Yaskawa INFORM job: DPRINT3D10.JBI

/JOB
//NAME DPRINT3D10
//POS
///NPOS 985,0,0,0,0,0
///TOOL 9
///POSTYPE PULSE
///PULSE
C00000=48313,52303,-120095,63672,-120169,-93276,0
C00001=48292,52332,-119999,63708,-120197,-93246,0
C00002=48271,52372,-119870,63749,-120237,-93206,0
C00003=48256,52403,-119767,63780,-120271,-93175,0
C00004=48247,52435,-119662,63805,-120306,-93144,0
C00005=48242,52474,-119535,63828,-120351,-93108,0
C00006=48240,52507,-119427,63845,-120390,-93077,0
C00007=48244,52540,-119319,63857,-120432,-93047,0
C00008=48254,52576,-119202,63863,-120480,-93015,0
C00009=48265,52610,-119093,63867,-120523,-92986,0
C00010=48282,52644,-118984,63864,-120571,-92958,0
C00011=48286,52651,-118962,63862,-120581,-92952,0
C00012=48302,52701,-118799,63868,-120646,-92909,0
C00013=30148,51851,-121170,60929,-120456,-93852,0
C00014=30162,51845,-121190,60911,-120453,-93859,0
C00015=30223,51818,-121280,60832,-120438,-93894,0
C00016=30294,51784,-121396,60738,-120418,-93935,0
C00017=30355,51745,-121525,60652,-120388,-93980,0
C00018=30411,51705,-121661,60572,-120352,-94026,0
C00019=30455,51662,-121806,60503,-120310,-94072,0
C00020=30494,51618,-121956,60440,-120263,-94119,0
C00021=30520,51571,-122113,60390,-120209,-94166,0
C00022=30539,51524,-122271,60346,-120151,-94213,0
C00023=30546,51477,-122432,60317,-120088,-94259,0
C00024=30545,51429,-122594,60295,-120021,-94303,0
C00025=30531,51382,-122754,60288,-119952,-94345,0
C00026=30511,51335,-122911,60290,-119880,-94386,0
C00027=30478,51291,-123064,60306,-119806,-94423,0
C00028=30438,51247,-123212,60330,-119733,-94459,0
C00029=30386,51206,-123350,60368,-119658,-94491,0
C00030=30328,51167,-123484,60415,-119583,-94519,0
C00031=30311,51158,-123514,60429,-119566,-94525,0
C00032=30263,51130,-123609,60469,-119511,-94545,0
C00033=30203,51101,-123709,60523,-119450,-94565,0
C00034=30111,51065,-123831,60608,-119369,-94586,0
C00035=30037,51041,-123911,60678,-119311,-94599,0
C00036=29931,51014,-124003,60783,-119238,-94610,0
C00037=29846,50997,-124062,60869,-119186,-94615,0
C00038=29731,50980,-124118,60989,-119124,-94615,0
C00039=29637,50970,-124150,61088,-119080,-94611,0
C00040=29518,50964,-124170,61217,-119032,-94601,0
C00041=29419,50962,-124173,61325,-118997,-94589,0
C00042=29301,50967,-124156,61458,-118964,-94568,0
C00043=29202,50974,-124127,61570,-118942,-94547,0
C00044=29088,50989,-124074,61703,-118925,-94516,0
C00045=29047,50995,-124051,61750,-118920,-94505,0
C00046=28992,51005,-124016,61816,-118916,-94487,0
C00047=28937,51018,-123970,61882,-118916,-94467,0
C00048=28868,51035,-123909,61966,-118916,-94441,0
C00049=28800,51055,-123840,62049,-118920,-94412,0
C00050=28711,51089,-123723,62163,-118936,-94367,0
C00051=28673,51104,-123669,62211,-118944,-94346,0
C00052=28632,51124,-123601,62266,-118957,-94322,0
C00053=28562,51163,-123464,62360,-118987,-94274,0
C00054=28530,51183,-123394,62404,-119003,-94249,0
C00055=28500,51205,-123319,62448,-119023,-94224,0
C00056=28479,51224,-123254,62479,-119041,-94203,0
C00057=28453,51251,-123161,62520,-119069,-94173,0
C00058=28414,51299,-122996,62585,-119119,-94121,0
C00059=28390,51349,-122825,62634,-119177,-94069,0
C00060=28372,51400,-122652,62677,-119238,-94017,0
C00061=28369,51452,-122476,62703,-119305,-93967,0
C00062=28374,51504,-122300,62722,-119375,-93918,0
C00063=28378,51516,-122258,62723,-119393,-93907,0
C00064=28393,51556,-122125,62724,-119449,-93871,0
C00065=28418,51607,-121954,62719,-119525,-93826,0
C00066=28461,51656,-121791,62695,-119603,-93786,0
C00067=28512,51703,-121635,62661,-119681,-93749,0
C00068=28543,51726,-121555,62637,-119724,-93731,0
C00069=28573,51746,-121489,62613,-119760,-93717,0
C00070=28645,51790,-121346,62555,-119842,-93686,0
C00071=28701,51817,-121255,62506,-119897,-93669,0
C00072=28759,51842,-121173,62453,-119950,-93654,0
C00073=28805,51861,-121111,62411,-119991,-93643,0
C00074=28853,51877,-121058,62366,-120029,-93635,0
C00075=28890,51889,-121021,62331,-120057,-93630,0
C00076=28990,51916,-120931,62234,-120128,-93618,0
C00077=29081,51935,-120870,62143,-120186,-93614,0
C00078=29190,51953,-120814,62031,-120248,-93614,0
C00079=29284,51962,-120783,61932,-120294,-93620,0
C00080=29399,51970,-120761,61809,-120344,-93630,0
C00081=29492,51970,-120760,61707,-120379,-93643,0
C00082=29608,51966,-120775,61579,-120415,-93664,0
C00083=29697,51959,-120803,61477,-120437,-93685,0
C00084=29810,51944,-120856,61345,-120458,-93715,0
C00085=29891,51928,-120908,61248,-120467,-93742,0
C00086=29997,51902,-120995,61120,-120471,-93782,0
C00087=30066,51881,-121068,61034,-120467,-93812,0
C00088=30146,51842,-121200,60928,-120443,-93860,0
C00089=25451,55201,-110574,67596,-122310,-90184,0
C00090=36364,52150,-120303,76476,-115314,-91905,0
C00091=38692,59001,-99858,76810,-121576,-86102,0
C00092=38615,59038,-99753,76902,-121554,-86062,0
C00093=38581,59057,-99701,76944,-121546,-86041,0
C00094=38542,59080,-99635,76993,-121538,-86017,0
C00095=38475,59130,-99497,77080,-121530,-85968,0
C00096=38443,59156,-99424,77123,-121528,-85943,0
C00097=38413,59183,-99346,77165,-121528,-85916,0
C00098=38391,59209,-99275,77197,-121531,-85893,0
C00099=38362,59245,-99174,77242,-121537,-85860,0
C00100=38317,59310,-98994,77314,-121551,-85802,0
C00101=38282,59379,-98800,77378,-121575,-85741,0
C00102=38253,59451,-98602,77437,-121602,-85680,0
C00103=38236,59525,-98397,77486,-121639,-85618,0
C00104=38224,59600,-98189,77530,-121679,-85557,0
C00105=38224,59618,-98139,77538,-121691,-85542,0
C00106=38225,59676,-97978,77562,-121728,-85496,0
C00107=38231,59753,-97768,77589,-121778,-85437,0
C00108=38251,59828,-97562,77602,-121838,-85380,0
C00109=38278,59901,-97362,77607,-121900,-85326,0
C00110=38297,59938,-97259,77605,-121935,-85300,0
C00111=38315,59970,-97171,77601,-121966,-85277,0
C00112=38360,60041,-96979,77587,-122037,-85228,0
C00113=38398,60086,-96854,77571,-122089,-85198,0
C00114=38438,60129,-96738,77550,-122139,-85170,0
C00115=38469,60162,-96650,77534,-122179,-85149,0
C00116=38503,60190,-96572,77514,-122218,-85131,0
C00117=38529,60211,-96516,77497,-122247,-85119,0
C00118=38602,60262,-96378,77448,-122323,-85090,0
C00119=38669,60299,-96278,77399,-122389,-85071,0
C00120=38752,60337,-96176,77335,-122463,-85053,0
C00121=38825,60362,-96109,77275,-122524,-85044,0
C00122=38914,60385,-96048,77198,-122594,-85039,0
C00123=38988,60396,-96017,77131,-122647,-85042,0
C00124=39082,60404,-95999,77043,-122710,-85050,0
C00125=39155,60403,-96003,76971,-122755,-85061,0
C00126=39249,60394,-96030,76875,-122808,-85083,0
C00127=39319,60380,-96067,76801,-122842,-85104,0
C00128=39410,60355,-96138,76701,-122883,-85137,0
C00129=39473,60331,-96204,76628,-122907,-85165,0
C00130=39557,60290,-96318,76527,-122932,-85210,0
C00131=39612,60258,-96406,76459,-122946,-85243,0
C00132=39678,60217,-96522,76375,-122960,-85286,0
C00133=39737,60168,-96657,76295,-122964,-85333,0
C00134=39792,60116,-96800,76218,-122964,-85382,0
C00135=39839,60058,-96960,76145,-122955,-85434,0
C00136=39881,59998,-97125,76076,-122941,-85488,0
C00137=39915,59933,-97303,76014,-122919,-85544,0
C00138=39943,59868,-97485,75956,-122893,-85600,0
C00139=39961,59799,-97674,75907,-122859,-85657,0
C00140=39974,59730,-97865,75863,-122821,-85713,0
C00141=39976,59660,-98058,75829,-122776,-85769,0
C00142=39973,59590,-98250,75801,-122728,-85823,0
C00143=39959,59521,-98440,75783,-122672,-85875,0
C00144=39940,59453,-98627,75772,-122616,-85926,0
C00145=39910,59389,-98806,75772,-122555,-85973,0
C00146=39875,59325,-98980,75778,-122492,-86018,0
C00147=39865,59311,-99021,75782,-122476,-86028,0
C00148=39835,59265,-99148,75791,-122426,-86060,0
C00149=39795,59216,-99283,75809,-122370,-86093,0
C00150=39733,59154,-99454,75843,-122292,-86133,0
C00151=39682,59111,-99571,75875,-122233,-86159,0
C00152=39606,59061,-99711,75928,-122154,-86188,0
C00153=39543,59026,-99805,75975,-122094,-86206,0
C00154=39457,58990,-99905,76045,-122018,-86223,0
C00155=39386,58966,-99971,76105,-121961,-86232,0
C00156=39293,58944,-100030,76188,-121892,-86236,0
C00157=39216,58931,-100063,76259,-121838,-86235,0
C00158=39120,58925,-100079,76352,-121777,-86225,0
C00159=39039,58925,-100077,76432,-121730,-86214,0
C00160=38945,58934,-100049,76530,-121681,-86192,0
C00161=38911,58939,-100035,76566,-121665,-86184,0
C00162=38864,58948,-100010,76617,-121642,-86170,0
C00163=38816,58961,-99973,76669,-121622,-86152,0
C00164=38771,58974,-99936,76720,-121604,-86136,0
C00165=38691,59038,-99755,76827,-121599,-86073,0
C00166=38691,58985,-99777,76837,-121614,-86054,0
C00167=29066,51891,-120835,62177,-120230,-93576,0
C00168=29144,51906,-120784,62099,-120279,-93573,0
C00169=29192,51914,-120759,62050,-120306,-93573,0
C00170=29275,51924,-120728,61964,-120349,-93577,0
C00171=29382,51934,-120697,61850,-120400,-93584,0
C00172=29408,51935,-120694,61823,-120411,-93587,0
C00173=29492,51937,-120689,61731,-120443,-93597,0
C00174=29601,51937,-120692,61611,-120483,-93614,0
C00175=29709,51929,-120719,61488,-120512,-93637,0
C00176=29816,51918,-120756,61365,-120536,-93663,0
C00177=29841,51915,-120769,61337,-120541,-93670,0
C00178=29919,51901,-120815,61244,-120551,-93694,0
C00179=29968,51891,-120850,61186,-120554,-93711,0
C00180=30019,51879,-120890,61124,-120558,-93729,0
C00181=30067,51865,-120937,61065,-120557,-93750,0
C00182=30111,51851,-120985,61010,-120553,-93769,0
C00183=30201,51818,-121097,60894,-120542,-93813,0
C00184=30258,51792,-121184,60819,-120527,-93846,0
C00185=30312,51764,-121277,60747,-120510,-93880,0
C00186=30351,51743,-121349,60694,-120495,-93905,0
C00187=30385,51721,-121422,60647,-120477,-93930,0
C00188=30409,51703,-121483,60612,-120461,-93950,0
C00189=30472,51651,-121655,60518,-120414,-94007,0
C00190=30501,51621,-121759,60472,-120383,-94040,0
C00191=30527,51587,-121870,60428,-120346,-94075,0
C00192=30547,51560,-121964,60393,-120317,-94103,0
C00193=30561,51532,-122059,60364,-120283,-94131,0
C00194=30576,51489,-122201,60329,-120230,-94173,0
C00195=30584,51460,-122300,60306,-120192,-94202,0
C00196=30586,51430,-122400,60289,-120153,-94229,0
C00197=30583,51390,-122537,60274,-120097,-94267,0
C00198=30579,51360,-122638,60265,-120053,-94294,0
C00199=30569,51330,-122740,60262,-120009,-94321,0
C00200=30549,51293,-122864,60267,-119951,-94352,0
C00201=30532,51263,-122965,60273,-119904,-94377,0
C00202=30508,51234,-123063,60285,-119856,-94401,0
C00203=30475,51202,-123172,60306,-119801,-94427,0
C00204=30445,51174,-123266,60327,-119751,-94449,0
C00205=30408,51147,-123358,60356,-119701,-94469,0
C00206=30365,51121,-123448,60391,-119650,-94488,0
C00207=30321,51096,-123533,60428,-119601,-94506,0
C00208=30272,51072,-123615,60471,-119550,-94521,0
C00209=30185,51035,-123739,60550,-119471,-94544,0
C00210=30103,51007,-123835,60629,-119403,-94560,0
C00211=30015,50981,-123923,60713,-119339,-94572,0
C00212=29922,50960,-123992,60807,-119279,-94579,0
C00213=29825,50943,-124051,60906,-119221,-94582,0
C00214=29724,50931,-124089,61012,-119172,-94579,0
C00215=29622,50922,-124118,61121,-119126,-94574,0
C00216=29518,50919,-124126,61235,-119088,-94561,0
C00217=29414,50920,-124123,61350,-119054,-94547,0
C00218=29311,50926,-124098,61466,-119030,-94526,0
C00219=29209,50936,-124063,61583,-119009,-94503,0
C00220=29112,50951,-124009,61697,-118997,-94474,0
C00221=29017,50969,-123943,61810,-118992,-94443,0
C00222=28929,50993,-123859,61918,-118995,-94408,0
C00223=28844,51020,-123766,62023,-119002,-94370,0
C00224=28758,51055,-123643,62134,-119021,-94324,0
C00225=28707,51078,-123564,62201,-119035,-94294,0
C00226=28662,51102,-123481,62261,-119053,-94265,0
C00227=28618,51127,-123394,62320,-119071,-94234,0
C00228=28580,51153,-123304,62374,-119093,-94204,0
C00229=28548,51181,-123210,62422,-119119,-94173,0
C00230=28514,51211,-123106,62473,-119148,-94138,0
C00231=28489,51240,-123007,62514,-119178,-94107,0
C00232=28469,51269,-122907,62548,-119210,-94076,0
C00233=28448,51305,-122785,62587,-119250,-94039,0
C00234=28437,51335,-122684,62614,-119285,-94008,0
C00235=28431,51365,-122582,62634,-119323,-93979,0
C00236=28425,51404,-122448,62658,-119372,-93941,0
C00237=28426,51434,-122347,62671,-119412,-93912,0
C00238=28433,51464,-122247,62677,-119454,-93884,0
C00239=28445,51506,-122106,62683,-119512,-93847,0
C00240=28458,51534,-122012,62681,-119554,-93822,0
C00241=28477,51563,-121915,62673,-119597,-93797,0
C00242=28507,51605,-121775,62659,-119663,-93761,0
C00243=28531,51631,-121688,62645,-119705,-93740,0
C00244=28561,51657,-121601,62624,-119749,-93720,0
C00245=28599,51689,-121496,62597,-119803,-93696,0
C00246=28643,51721,-121390,62563,-119860,-93672,0
C00247=28717,51764,-121249,62502,-119942,-93643,0
C00248=28750,51781,-121192,62474,-119975,-93632,0
C00249=28790,51800,-121130,62439,-120014,-93620,0
C00250=28836,51818,-121070,62396,-120055,-93609,0
C00251=28900,51842,-120990,62338,-120109,-93596,0
C00252=28965,51864,-120920,62276,-120160,-93585,0
C00253=28974,51867,-120912,62267,-120166,-93585,0
C00254=29068,51902,-120798,62180,-120245,-93566,0
C00255=39943,50914,-124372,72212,-115599,-93497,0
C00256=35334,54043,-114097,78273,-116418,-89868,0
C00257=36297,54454,-112860,77429,-117185,-89597,0
C00258=40949,51295,-123088,71276,-116378,-93209,0
C00259=40026,50945,-124269,72134,-115663,-93473,0
C00260=35605,54738,-111986,78248,-117048,-89258,0
C00261=36478,55133,-110816,77500,-117769,-89005,0
C00262=42177,51262,-123232,69935,-116794,-93388,0
C00263=33602,54748,-111917,58580,-125515,-91919,0
C00264=34233,54163,-113709,79451,-115969,-89637,0
C00265=35135,54535,-112592,78656,-116671,-89391,0
C00266=34900,54747,-111946,78974,-116702,-89171,0
C00267=35368,54950,-111341,78569,-117079,-89039,0
C00268=35551,54786,-111840,78321,-117055,-89209,0
C00269=36110,54506,-112698,77641,-117132,-89528,0
C00270=34834,55007,-111160,57349,-126335,-91958,0
C00271=36863,53301,-116438,54206,-124911,-93686,0
C00272=39303,53272,-116584,73829,-117628,-91057,0
C00273=44071,55812,-108960,69905,-122100,-89467,0
C00274=34853,54989,-111215,79109,-116844,-88946,0
C00275=33011,56887,-105605,81638,-117037,-87071,0
C00276=36074,54033,-114146,77503,-116763,-89961,0
C00277=40139,51272,-123147,72141,-116051,-93140,0
C00278=48385,52777,-118383,63852,-120867,-92777,0
C00279=48412,52795,-118324,63830,-120899,-92765,0
C00280=48487,52840,-118184,63770,-120980,-92737,0
C00281=48544,52867,-118098,63720,-121034,-92721,0
C00282=48600,52891,-118023,63670,-121084,-92709,0
C00283=48648,52910,-117962,63626,-121126,-92699,0
C00284=48698,52927,-117910,63579,-121165,-92691,0
C00285=48776,52949,-117842,63505,-121220,-92684,0
C00286=48831,52963,-117798,63452,-121258,-92680,0
C00287=48887,52975,-117762,63396,-121293,-92678,0
C00288=48966,52987,-117724,63315,-121339,-92680,0
C00289=49026,52996,-117698,63254,-121373,-92681,0
C00290=49087,53002,-117682,63189,-121403,-92686,0
C00291=49164,53006,-117671,63107,-121437,-92695,0
C00292=49227,53008,-117665,63039,-121465,-92703,0
C00293=49291,53007,-117669,62969,-121488,-92713,0
C00294=49363,53003,-117684,62888,-121511,-92728,0
C00295=49427,52999,-117699,62816,-121530,-92742,0
C00296=49490,52991,-117725,62743,-121545,-92759,0
C00297=49555,52981,-117761,62667,-121557,-92779,0
C00298=49617,52970,-117799,62593,-121567,-92799,0
C00299=49678,52955,-117846,62519,-121574,-92822,0
C00300=49777,52928,-117936,62398,-121578,-92861,0
C00301=49856,52900,-118025,62298,-121575,-92898,0
C00302=49946,52864,-118146,62182,-121563,-92945,0
C00303=50004,52833,-118246,62103,-121548,-92982,0
C00304=50069,52795,-118370,62013,-121525,-93026,0
C00305=50124,52753,-118507,61933,-121493,-93072,0
C00306=50173,52709,-118650,61858,-121458,-93119,0
C00307=50211,52662,-118802,61794,-121414,-93167,0
C00308=50244,52614,-118958,61735,-121366,-93215,0
C00309=50263,52564,-119119,61690,-121311,-93263,0
C00310=50277,52514,-119283,61651,-121252,-93310,0
C00311=50277,52463,-119448,61626,-121189,-93356,0
C00312=50272,52413,-119612,61609,-121122,-93400,0
C00313=50253,52363,-119773,61606,-121053,-93442,0
C00314=50228,52314,-119932,61611,-120982,-93482,0
C00315=50186,52261,-120104,61632,-120899,-93523,0
C00316=50157,52229,-120210,61649,-120847,-93548,0
C00317=50124,52200,-120306,61671,-120798,-93570,0
C00318=50088,52170,-120403,61696,-120748,-93592,0
C00319=50049,52143,-120491,61726,-120698,-93611,0
C00320=50006,52117,-120574,61763,-120650,-93627,0
C00321=49957,52090,-120662,61804,-120598,-93645,0
C00322=49908,52067,-120736,61847,-120551,-93658,0
C00323=49856,52047,-120800,61895,-120507,-93669,0
C00324=49793,52024,-120876,61954,-120454,-93681,0
C00325=49737,52007,-120930,62007,-120413,-93688,0
C00326=49680,51993,-120976,62064,-120374,-93692,0
C00327=49604,51975,-121033,62139,-120326,-93697,0
C00328=49545,51964,-121067,62199,-120290,-93698,0
C00329=49483,51956,-121092,62263,-120258,-93697,0
C00330=49397,51946,-121124,62353,-120214,-93693,0
C00331=49337,51941,-121138,62417,-120188,-93689,0
C00332=49275,51939,-121144,62484,-120163,-93681,0
C00333=49182,51937,-121147,62586,-120128,-93669,0
C00334=49123,51938,-121142,62651,-120109,-93659,0
C00335=49063,51942,-121127,62719,-120093,-93646,0
C00336=48988,51948,-121106,62804,-120073,-93630,0
C00337=48912,51956,-121075,62892,-120057,-93610,0
C00338=48805,51975,-121011,63018,-120042,-93577,0
C00339=48760,51984,-120980,63071,-120037,-93562,0
C00340=48707,51997,-120936,63136,-120035,-93542,0
C00341=48615,52024,-120843,63249,-120036,-93503,0
C00342=48572,52038,-120793,63303,-120038,-93483,0
C00343=48528,52055,-120737,63360,-120043,-93461,0
C00344=48453,52089,-120622,63457,-120059,-93418,0
C00345=48394,52123,-120512,63537,-120079,-93379,0
C00346=48365,52142,-120445,63579,-120093,-93356,0
C00347=48320,52178,-120328,63644,-120120,-93316,0
C00348=48268,52225,-120171,63723,-120159,-93265,0
C00349=48259,52237,-120133,63739,-120169,-93252,0
C00350=48230,52276,-120004,63788,-120206,-93212,0
C00351=48197,52328,-119833,63848,-120258,-93159,0
C00352=48180,52381,-119657,63892,-120317,-93107,0
C00353=48169,52436,-119478,63930,-120379,-93054,0
C00354=48169,52449,-119435,63935,-120395,-93043,0
C00355=48172,52491,-119298,63952,-120446,-93005,0
C00356=48177,52518,-119212,63958,-120480,-92981,0
C00357=48185,52546,-119120,63963,-120517,-92956,0
C00358=48198,52574,-119031,63961,-120556,-92933,0
C00359=48213,52600,-118947,63957,-120591,-92911,0
C00360=48250,52655,-118771,63942,-120672,-92867,0
C00361=48284,52691,-118655,63922,-120727,-92839,0
C00362=48322,52727,-118542,63897,-120783,-92813,0
C00363=48328,52732,-118524,63893,-120792,-92809,0
C00364=48363,52780,-118371,63877,-120862,-92771,0
C00365=39595,59020,-99695,75955,-122172,-86157,0
C00366=39524,58985,-99793,76010,-122107,-86175,0
C00367=39448,58957,-99869,76074,-122043,-86186,0
C00368=39369,58933,-99934,76141,-121981,-86194,0
C00369=39287,58918,-99974,76216,-121923,-86194,0
C00370=39205,58907,-100002,76293,-121867,-86190,0
C00371=39121,58906,-100005,76376,-121816,-86179,0
C00372=39038,58909,-99994,76460,-121769,-86165,0
C00373=38956,58921,-99960,76547,-121729,-86143,0
C00374=38875,58937,-99913,76634,-121692,-86119,0
C00375=38798,58962,-99841,76721,-121663,-86087,0
C00376=38723,58991,-99759,76808,-121638,-86053,0
C00377=38644,59033,-99641,76905,-121617,-86008,0
C00378=38596,59061,-99563,76964,-121607,-85979,0
C00379=38554,59090,-99480,77019,-121601,-85950,0
C00380=38512,59122,-99392,77074,-121597,-85918,0
C00381=38474,59155,-99299,77126,-121596,-85886,0
C00382=38440,59191,-99198,77175,-121598,-85853,0
C00383=38404,59231,-99087,77227,-121602,-85816,0
C00384=38375,59270,-98979,77273,-121609,-85780,0
C00385=38351,59310,-98867,77313,-121621,-85745,0
C00386=38324,59359,-98731,77361,-121636,-85702,0
C00387=38306,59401,-98616,77397,-121651,-85667,0
C00388=38292,59444,-98497,77429,-121670,-85631,0
C00389=38276,59500,-98342,77468,-121696,-85584,0
C00390=38269,59542,-98224,77494,-121717,-85549,0
C00391=38266,59586,-98103,77516,-121744,-85513,0
C00392=38263,59647,-97934,77545,-121781,-85465,0
C00393=38265,59690,-97818,77561,-121808,-85432,0
C00394=38273,59733,-97699,77573,-121839,-85398,0
C00395=38285,59797,-97524,77588,-121886,-85350,0
C00396=38297,59837,-97413,77594,-121919,-85320,0
C00397=38313,59878,-97302,77596,-121954,-85290,0
C00398=38334,59928,-97165,77597,-121998,-85253,0
C00399=38361,59978,-97027,77593,-122046,-85217,0
C00400=38408,60048,-96836,77577,-122118,-85169,0
C00401=38430,60077,-96759,77568,-122149,-85150,0
C00402=38457,60108,-96673,77556,-122185,-85129,0
C00403=38489,60140,-96587,77539,-122225,-85109,0
C00404=38533,60182,-96473,77514,-122278,-85083,0
C00405=38579,60221,-96368,77485,-122331,-85059,0
C00406=38653,60270,-96235,77436,-122407,-85032,0
C00407=38711,60301,-96151,77393,-122462,-85015,0
C00408=38747,60318,-96106,77365,-122495,-85008,0
C00409=38811,60341,-96042,77313,-122549,-84999,0
C00410=38894,60368,-95971,77244,-122618,-84990,0
C00411=38914,60372,-95960,77226,-122633,-84990,0
C00412=38981,60384,-95928,77167,-122683,-84990,0
C00413=39068,60397,-95897,77087,-122745,-84994,0
C00414=39157,60398,-95894,77001,-122801,-85006,0
C00415=39245,60395,-95905,76914,-122854,-85022,0
C00416=39266,60392,-95913,76892,-122864,-85028,0
C00417=39332,60381,-95943,76823,-122899,-85046,0
C00418=39373,60372,-95969,76778,-122918,-85060,0
C00419=39417,60361,-96001,76730,-122939,-85075,0
C00420=39459,60346,-96042,76682,-122955,-85093,0
C00421=39498,60330,-96086,76637,-122969,-85111,0
C00422=39579,60293,-96190,76541,-122995,-85152,0
C00423=39631,60261,-96277,76475,-123008,-85185,0
C00424=39681,60227,-96371,76411,-123017,-85219,0
C00425=39718,60201,-96443,76363,-123023,-85245,0
C00426=39750,60173,-96520,76319,-123025,-85272,0
C00427=39775,60150,-96584,76284,-123025,-85294,0
C00428=39839,60082,-96770,76191,-123021,-85356,0
C00429=39870,60041,-96885,76141,-123013,-85393,0
C00430=39899,59996,-97009,76092,-123001,-85433,0
C00431=39922,59957,-97114,76051,-122990,-85467,0
C00432=39942,59919,-97221,76015,-122976,-85500,0
C00433=39964,59859,-97386,75965,-122950,-85550,0
C00434=39979,59817,-97501,75932,-122932,-85586,0
C00435=39989,59774,-97618,75902,-122910,-85621,0
C00436=39998,59715,-97780,75867,-122876,-85668,0
C00437=40003,59671,-97902,75842,-122849,-85704,0
C00438=40003,59626,-98026,75822,-122821,-85739,0
C00439=39998,59571,-98178,75802,-122780,-85781,0
C00440=39992,59526,-98303,75787,-122747,-85816,0
C00441=39981,59481,-98426,75778,-122710,-85850,0
C00442=39964,59431,-98564,75772,-122667,-85887,0
C00443=39948,59387,-98685,75768,-122628,-85920,0
C00444=39927,59344,-98804,75770,-122586,-85950,0
C00445=39900,59301,-98922,75777,-122541,-85980,0
C00446=39873,59260,-99036,75786,-122498,-86009,0
C00447=39841,59220,-99146,75800,-122452,-86036,0
C00448=39783,59157,-99318,75830,-122375,-86077,0
C00449=39725,59107,-99456,75864,-122307,-86108,0
C00450=39665,59062,-99582,75903,-122241,-86135,0
C00451=39599,58976,-99818,75931,-122145,-86193,0
C00452=23775,60523,-95311,71968,-125942,-85610,0
C00453=23816,60447,-95518,71888,-125912,-85675,0
C00454=23839,60389,-95677,71836,-125882,-85723,0
C00455=23861,60320,-95866,71779,-125844,-85780,0
C00456=23873,60249,-96060,71731,-125798,-85836,0
C00457=23879,60177,-96256,71689,-125749,-85892,0
C00458=23875,60105,-96451,71657,-125693,-85946,0
C00459=23866,60034,-96646,71631,-125634,-85998,0
C00460=23846,59965,-96835,71616,-125571,-86048,0
C00461=23820,59897,-97020,71608,-125504,-86095,0
C00462=23785,59833,-97196,71611,-125435,-86138,0
C00463=23745,59771,-97365,71621,-125365,-86179,0
C00464=23696,59715,-97521,71642,-125292,-86214,0
C00465=23643,59661,-97668,71669,-125221,-86246,0
C00466=23574,59607,-97815,71712,-125140,-86276,0
C00467=23529,59575,-97902,71742,-125089,-86293,0
C00468=23450,59528,-98030,71799,-125007,-86315,0
C00469=23388,59499,-98110,71847,-124949,-86327,0
C00470=23299,59467,-98198,71921,-124873,-86337,0
C00471=23230,59448,-98249,71982,-124818,-86340,0
C00472=23135,59432,-98293,72069,-124750,-86337,0
C00473=23061,59424,-98312,72140,-124701,-86330,0
C00474=22966,59424,-98311,72236,-124645,-86314,0
C00475=22889,59430,-98295,72316,-124604,-86297,0
C00476=22797,59446,-98249,72417,-124562,-86269,0
C00477=22721,59465,-98197,72502,-124532,-86242,0
C00478=22635,59496,-98109,72604,-124503,-86203,0
C00479=22563,59528,-98020,72691,-124485,-86167,0
C00480=22487,59573,-97895,72790,-124472,-86119,0
C00481=22458,59592,-97843,72828,-124470,-86099,0
C00482=22423,59618,-97772,72875,-124467,-86074,0
C00483=22389,59648,-97688,72924,-124468,-86045,0
C00484=22346,59688,-97578,72986,-124472,-86007,0
C00485=22306,59731,-97459,73047,-124480,-85967,0
C00486=22257,59798,-97273,73129,-124498,-85907,0
C00487=22236,59830,-97186,73165,-124510,-85878,0
C00488=22216,59866,-97087,73203,-124522,-85848,0
C00489=22186,59934,-96900,73265,-124554,-85790,0
C00490=22167,59996,-96731,73314,-124586,-85740,0
C00491=22160,60031,-96635,73338,-124606,-85711,0
C00492=22152,60091,-96471,73375,-124645,-85664,0
C00493=22147,60169,-96257,73417,-124697,-85603,0
C00494=22149,60187,-96208,73425,-124711,-85589,0
C00495=22155,60247,-96044,73448,-124757,-85544,0
C00496=22167,60325,-95832,73473,-124820,-85486,0
C00497=22192,60401,-95625,73486,-124888,-85432,0
C00498=22221,60475,-95423,73493,-124959,-85380,0
C00499=22230,60492,-95377,73492,-124976,-85368,0
C00500=22261,60546,-95231,73488,-125033,-85332,0
C00501=22283,60579,-95141,73482,-125069,-85311,0
C00502=22308,60613,-95049,73474,-125109,-85289,0
C00503=22336,60645,-94962,73461,-125149,-85269,0
C00504=22365,60674,-94884,73447,-125187,-85252,0
C00505=22429,60733,-94725,73413,-125267,-85217,0
C00506=22478,60769,-94627,73383,-125323,-85198,0
C00507=22529,60803,-94537,73348,-125379,-85181,0
C00508=22569,60827,-94472,73321,-125420,-85170,0
C00509=22608,60847,-94418,73292,-125458,-85161,0
C00510=22625,60855,-94398,73279,-125474,-85158,0
C00511=22680,60877,-94337,73236,-125523,-85151,0
C00512=22725,60895,-94291,73200,-125564,-85145,0
C00513=22769,60908,-94256,73163,-125600,-85143,0
C00514=22801,60915,-94236,73135,-125626,-85143,0
C00515=22890,60933,-94190,73055,-125693,-85144,0
C00516=22967,60940,-94172,72982,-125746,-85152,0
C00517=23059,60941,-94170,72892,-125804,-85167,0
C00518=23134,60934,-94190,72814,-125845,-85186,0
C00519=23224,60918,-94233,72716,-125890,-85213,0
C00520=23295,60899,-94286,72637,-125920,-85240,0
C00521=23381,60867,-94374,72534,-125951,-85279,0
C00522=23444,60837,-94457,72457,-125967,-85314,0
C00523=23522,60790,-94585,72355,-125982,-85363,0
C00524=23576,60750,-94693,72281,-125987,-85402,0
C00525=23644,60689,-94858,72183,-125983,-85460,0
C00526=23680,60651,-94963,72128,-125977,-85496,0
C00527=23732,60587,-95137,72043,-125962,-85553,0
C00528=23825,60523,-95313,71917,-125973,-85619,0
C00529=25489,55155,-110561,67572,-122361,-90161,0
C00530=36365,52089,-120325,76484,-115334,-91883,0
C00531=36365,52027,-120346,76491,-115352,-91861,0
C00532=23826,60495,-95267,71941,-126008,-85582,0
C00533=23863,60420,-95471,71866,-125976,-85646,0
C00534=23883,60366,-95619,71819,-125947,-85690,0
C00535=23897,60314,-95762,71778,-125918,-85733,0
C00536=23908,60271,-95878,71746,-125892,-85767,0
C00537=23914,60229,-95993,71718,-125865,-85801,0
C00538=23917,60163,-96173,71681,-125818,-85851,0
C00539=23918,60119,-96294,71658,-125785,-85885,0
C00540=23915,60075,-96412,71640,-125751,-85918,0
C00541=23904,60014,-96580,71620,-125698,-85963,0
C00542=23895,59969,-96701,71607,-125660,-85995,0
C00543=23881,59926,-96819,71599,-125619,-86026,0
C00544=23858,59871,-96969,71595,-125565,-86063,0
C00545=23839,59829,-97085,71593,-125521,-86092,0
C00546=23815,59788,-97197,71597,-125476,-86120,0
C00547=23782,59741,-97325,71607,-125421,-86150,0
C00548=23753,59702,-97431,71617,-125375,-86175,0
C00549=23719,59666,-97531,71633,-125327,-86197,0
C00550=23678,59628,-97634,71655,-125275,-86219,0
C00551=23640,59595,-97726,71677,-125227,-86238,0
C00552=23597,59563,-97811,71705,-125178,-86255,0
C00553=23552,59536,-97886,71737,-125130,-86268,0
C00554=23505,59509,-97959,71771,-125083,-86280,0
C00555=23455,59486,-98023,71810,-125036,-86290,0
C00556=23372,59449,-98122,71876,-124960,-86304,0
C00557=23295,59426,-98185,71943,-124897,-86309,0
C00558=23215,59407,-98236,72014,-124836,-86310,0
C00559=23133,59398,-98262,72091,-124781,-86304,0
C00560=23051,59393,-98275,72172,-124728,-86294,0
C00561=22969,59397,-98262,72257,-124683,-86277,0
C00562=22887,59406,-98236,72343,-124642,-86256,0
C00563=22808,59424,-98186,72432,-124609,-86229,0
C00564=22730,59446,-98123,72521,-124579,-86199,0
C00565=22656,59477,-98037,72610,-124558,-86163,0
C00566=22586,59512,-97940,72698,-124542,-86124,0
C00567=22521,59555,-97821,72784,-124535,-86080,0
C00568=22460,59602,-97692,72868,-124533,-86033,0
C00569=22406,59655,-97545,72947,-124540,-85983,0
C00570=22357,59711,-97390,73024,-124551,-85932,0
C00571=22314,59771,-97225,73096,-124568,-85878,0
C00572=22282,59824,-97081,73153,-124587,-85832,0
C00573=22246,59901,-96867,73227,-124620,-85766,0
C00574=22226,59961,-96705,73275,-124651,-85718,0
C00575=22208,60043,-96481,73332,-124698,-85651,0
C00576=22202,60107,-96306,73370,-124740,-85602,0
C00577=22203,60190,-96078,73408,-124801,-85538,0
C00578=22211,60256,-95899,73433,-124851,-85488,0
C00579=22231,60337,-95678,73452,-124921,-85429,0
C00580=22254,60403,-95500,73462,-124981,-85383,0
C00581=22291,60479,-95292,73462,-125058,-85331,0
C00582=22328,60542,-95123,73456,-125124,-85289,0
C00583=22381,60610,-94938,73437,-125204,-85246,0
C00584=22402,60634,-94873,73429,-125234,-85231,0
C00585=22432,60666,-94786,73414,-125275,-85212,0
C00586=22466,60697,-94704,73395,-125318,-85194,0
C00587=22511,60735,-94601,73369,-125373,-85173,0
C00588=22560,60772,-94503,73339,-125428,-85154,0
C00589=22637,60817,-94381,73285,-125507,-85132,0
C00590=22671,60835,-94332,73260,-125542,-85124,0
C00591=22710,60853,-94284,73231,-125579,-85117,0
C00592=22754,60869,-94241,73196,-125616,-85112,0
C00593=22815,60890,-94185,73146,-125669,-85107,0
C00594=22875,60907,-94140,73095,-125719,-85104,0
C00595=22898,60911,-94129,73074,-125736,-85105,0
C00596=22964,60920,-94107,73013,-125783,-85110,0
C00597=23051,60925,-94093,72929,-125842,-85121,0
C00598=23138,60920,-94107,72841,-125891,-85140,0
C00599=23225,60911,-94134,72750,-125938,-85162,0
C00600=23309,60891,-94190,72656,-125976,-85192,0
C00601=23392,60866,-94258,72561,-126010,-85226,0
C00602=23470,60831,-94353,72465,-126034,-85266,0
C00603=23530,60801,-94435,72391,-126049,-85299,0
C00604=23547,60792,-94460,72370,-126052,-85308,0
C00605=23600,60755,-94561,72298,-126059,-85346,0
C00606=23681,60686,-94749,72182,-126059,-85412,0
C00607=23722,60642,-94867,72119,-126052,-85452,0
C00608=23760,60595,-94994,72058,-126041,-85495,0
C00609=23786,60561,-95088,72013,-126032,-85526,0
C00610=23870,60492,-95275,71895,-126032,-85592,0
C00611=35334,53985,-114119,78281,-116434,-89847,0
C00612=36297,54396,-112881,77437,-117202,-89576,0
C00613=40949,51232,-123110,71284,-116401,-93187,0
C00614=39943,50850,-124394,72219,-115622,-93474,0
C00615=35389,53938,-114263,78207,-116427,-89896,0
C00616=35605,54680,-112007,78256,-117064,-89238,0
C00617=36478,55075,-110837,77509,-117786,-88984,0
C00618=42177,51198,-123255,69943,-116819,-93367,0
C00619=33602,54690,-111938,58591,-125543,-91901,0
C00620=34234,54104,-113731,79458,-115985,-89616,0
C00621=35135,54477,-112613,78664,-116688,-89370,0
C00622=34900,54689,-111967,78982,-116717,-89150,0
C00623=35368,54893,-111362,78577,-117094,-89018,0
C00624=35551,54728,-111861,78329,-117071,-89188,0
C00625=36111,54448,-112720,77649,-117148,-89507,0
C00626=34834,54950,-111182,57360,-126362,-91940,0
C00627=36849,53253,-116426,54239,-124952,-93657,0
C00628=39303,53212,-116606,73837,-117647,-91036,0
C00629=44041,55737,-109037,69939,-122090,-89459,0
C00630=34854,54932,-111236,79117,-116860,-88925,0
C00631=33023,56818,-105666,81630,-117048,-87064,0
C00632=36074,53974,-114167,77511,-116781,-89940,0
C00633=40139,51208,-123170,72148,-116073,-93118,0
C00634=48465,52781,-118198,63805,-121000,-92712,0
C00635=48541,52824,-118061,63742,-121081,-92684,0
C00636=48579,52844,-118000,63710,-121118,-92673,0
C00637=48620,52863,-117940,63674,-121157,-92662,0
C00638=48663,52879,-117890,63635,-121192,-92655,0
C00639=48709,52895,-117840,63592,-121228,-92648,0
C00640=48802,52924,-117752,63504,-121298,-92637,0
C00641=48901,52945,-117686,63406,-121361,-92633,0
C00642=49001,52964,-117630,63304,-121422,-92633,0
C00643=49106,52975,-117597,63195,-121476,-92640,0
C00644=49211,52983,-117575,63084,-121525,-92649,0
C00645=49317,52983,-117576,62968,-121567,-92666,0
C00646=49399,52981,-117586,62877,-121596,-92681,0
C00647=49423,52980,-117590,62850,-121604,-92686,0
C00648=49475,52975,-117607,62791,-121617,-92699,0
C00649=49526,52968,-117630,62732,-121630,-92713,0
C00650=49627,52951,-117685,62613,-121648,-92743,0
C00651=49677,52940,-117723,62552,-121654,-92762,0
C00652=49722,52929,-117761,62498,-121658,-92779,0
C00653=49814,52902,-117848,62384,-121661,-92817,0
C00654=49861,52885,-117902,62325,-121658,-92840,0
C00655=49898,52870,-117952,62276,-121654,-92859,0
C00656=49983,52833,-118073,62166,-121640,-92905,0
C00657=50036,52804,-118169,62094,-121624,-92940,0
C00658=50082,52774,-118264,62029,-121606,-92973,0
C00659=50118,52750,-118343,61977,-121590,-93001,0
C00660=50150,52725,-118425,61931,-121570,-93028,0
C00661=50192,52683,-118558,61864,-121536,-93071,0
C00662=50220,52655,-118650,61821,-121512,-93101,0
C00663=50242,52627,-118742,61783,-121484,-93130,0
C00664=50267,52584,-118880,61735,-121440,-93172,0
C00665=50283,52553,-118980,61702,-121408,-93202,0
C00666=50294,52522,-119082,61675,-121373,-93231,0
C00667=50302,52481,-119217,61647,-121324,-93270,0
C00668=50307,52448,-119323,61626,-121284,-93299,0
C00669=50306,52415,-119428,61612,-121243,-93328,0
C00670=50298,52376,-119555,61602,-121191,-93363,0
C00671=50290,52343,-119662,61595,-121146,-93390,0
C00672=50275,52311,-119767,61596,-121100,-93418,0
C00673=50254,52276,-119881,61603,-121047,-93446,0
C00674=50233,52244,-119984,61611,-120999,-93472,0
C00675=50205,52212,-120087,61627,-120950,-93495,0
C00676=50173,52182,-120183,61648,-120900,-93518,0
C00677=50138,52153,-120280,61672,-120850,-93540,0
C00678=50098,52124,-120373,61703,-120799,-93559,0
C00679=50030,52079,-120520,61756,-120716,-93590,0
C00680=49960,52043,-120636,61817,-120645,-93612,0
C00681=49884,52009,-120744,61885,-120576,-93631,0
C00682=49800,51981,-120835,61964,-120510,-93644,0
C00683=49713,51956,-120916,62048,-120446,-93654,0
C00684=49620,51936,-120979,62142,-120389,-93658,0
C00685=49525,51920,-121030,62239,-120334,-93659,0
C00686=49426,51910,-121061,62344,-120286,-93653,0
C00687=49326,51903,-121081,62451,-120242,-93645,0
C00688=49225,51902,-121080,62561,-120205,-93630,0
C00689=49124,51905,-121068,62673,-120173,-93612,0
C00690=49026,51914,-121034,62786,-120150,-93589,0
C00691=48929,51927,-120989,62898,-120132,-93563,0
C00692=48837,51946,-120924,63008,-120122,-93531,0
C00693=48747,51968,-120850,63117,-120118,-93498,0
C00694=48662,51993,-120762,63222,-120119,-93461,0
C00695=48595,52017,-120682,63307,-120125,-93429,0
C00696=48507,52056,-120552,63421,-120141,-93379,0
C00697=48449,52088,-120446,63499,-120159,-93342,0
C00698=48380,52134,-120292,63596,-120191,-93288,0
C00699=48335,52172,-120166,63664,-120221,-93247,0
C00700=48287,52225,-119994,63741,-120267,-93191,0
C00701=48256,52268,-119851,63794,-120309,-93146,0
C00702=48230,52324,-119667,63849,-120367,-93090,0
C00703=48217,52371,-119513,63885,-120419,-93045,0
C00704=48214,52430,-119325,63916,-120488,-92992,0
C00705=48219,52479,-119165,63933,-120548,-92947,0
C00706=48238,52536,-118980,63939,-120623,-92898,0
C00707=48247,52557,-118912,63939,-120652,-92880,0
C00708=48262,52586,-118822,63935,-120691,-92857,0
C00709=48283,52615,-118727,63926,-120734,-92833,0
C00710=48311,52651,-118611,63912,-120788,-92805,0
C00711=48345,52688,-118494,63892,-120844,-92777,0
C00712=48404,52738,-118335,63851,-120926,-92741,0
C00713=48460,52782,-118195,63811,-120999,-92710,0
C00714=39767,59019,-99575,75817,-122324,-86123,0
C00715=39694,58969,-99712,75868,-122248,-86152,0
C00716=39640,58939,-99794,75909,-122195,-86168,0
C00717=39585,58914,-99863,75952,-122147,-86179,0
C00718=39541,58894,-99917,75988,-122107,-86189,0
C00719=39495,58879,-99960,76026,-122070,-86195,0
C00720=39422,58859,-100014,76089,-122014,-86200,0
C00721=39373,58847,-100047,76133,-121976,-86202,0
C00722=39323,58838,-100069,76179,-121941,-86202,0
C00723=39251,58831,-100087,76248,-121894,-86197,0
C00724=39199,58827,-100097,76298,-121861,-86192,0
C00725=39146,58827,-100096,76350,-121830,-86185,0
C00726=39078,58832,-100082,76420,-121793,-86171,0
C00727=39025,58837,-100068,76475,-121765,-86159,0
C00728=38973,58845,-100042,76531,-121740,-86145,0
C00729=38911,58860,-100000,76598,-121713,-86124,0
C00730=38859,58874,-99961,76656,-121692,-86105,0
C00731=38808,58892,-99910,76714,-121674,-86084,0
C00732=38756,58915,-99845,76776,-121657,-86058,0
C00733=38707,58937,-99782,76834,-121643,-86033,0
C00734=38661,58964,-99707,76891,-121632,-86005,0
C00735=38618,58993,-99625,76946,-121627,-85975,0
C00736=38575,59024,-99538,77002,-121621,-85944,0
C00737=38536,59058,-99443,77055,-121620,-85911,0
C00738=38474,59116,-99282,77142,-121619,-85857,0
C00739=38427,59172,-99124,77212,-121628,-85805,0
C00740=38386,59232,-98958,77278,-121640,-85751,0
C00741=38354,59296,-98781,77337,-121662,-85696,0
C00742=38328,59361,-98599,77391,-121688,-85640,0
C00743=38312,59430,-98410,77436,-121721,-85584,0
C00744=38301,59499,-98220,77477,-121758,-85527,0
C00745=38301,59569,-98027,77507,-121802,-85472,0
C00746=38307,59639,-97834,77531,-121850,-85417,0
C00747=38323,59708,-97644,77546,-121902,-85365,0
C00748=38344,59777,-97457,77554,-121958,-85314,0
C00749=38376,59842,-97278,77552,-122017,-85267,0
C00750=38412,59906,-97103,77545,-122079,-85222,0
C00751=38457,59965,-96941,77526,-122145,-85182,0
C00752=38489,60003,-96839,77511,-122187,-85157,0
C00753=38507,60023,-96786,77503,-122210,-85144,0
C00754=38570,60083,-96620,77468,-122287,-85106,0
C00755=38611,60118,-96527,77443,-122335,-85085,0
C00756=38654,60148,-96446,77414,-122379,-85068,0
C00757=38700,60178,-96363,77383,-122426,-85051,0
C00758=38746,60204,-96294,77349,-122471,-85037,0
C00759=38794,60226,-96235,77312,-122515,-85027,0
C00760=38849,60250,-96172,77269,-122564,-85017,0
C00761=38899,60267,-96126,77228,-122606,-85011,0
C00762=38949,60280,-96092,77185,-122645,-85008,0
C00763=39012,60294,-96054,77129,-122693,-85007,0
C00764=39063,60302,-96033,77084,-122730,-85008,0
C00765=39114,60306,-96023,77035,-122764,-85013,0
C00766=39183,60310,-96015,76970,-122809,-85020,0
C00767=39233,60309,-96018,76921,-122839,-85028,0
C00768=39283,60304,-96032,76870,-122868,-85040,0
C00769=39355,60295,-96058,76795,-122907,-85058,0
C00770=39402,60286,-96084,76745,-122930,-85072,0
C00771=39449,60272,-96121,76693,-122950,-85089,0
C00772=39506,60255,-96169,76630,-122975,-85111,0
C00773=39564,60234,-96229,76563,-122998,-85137,0
C00774=39644,60194,-96338,76467,-123022,-85180,0
C00775=39675,60177,-96386,76428,-123030,-85198,0
C00776=39712,60154,-96449,76382,-123038,-85221,0
C00777=39749,60127,-96524,76333,-123044,-85249,0
C00778=39797,60090,-96626,76270,-123048,-85285,0
C00779=39842,60050,-96736,76208,-123050,-85322,0
C00780=39911,59972,-96950,76104,-123042,-85394,0
C00781=39943,59929,-97068,76053,-123034,-85432,0
C00782=39955,59910,-97122,76032,-123029,-85449,0
C00783=39985,59853,-97278,75977,-123009,-85498,0
C00784=40009,59798,-97429,75928,-122988,-85545,0
C00785=40016,59781,-97476,75913,-122981,-85560,0
C00786=40036,59706,-97682,75860,-122944,-85621,0
C00787=40050,59631,-97891,75811,-122902,-85683,0
C00788=40053,59554,-98101,75774,-122853,-85743,0
C00789=40049,59478,-98311,75743,-122800,-85803,0
C00790=40034,59403,-98518,75724,-122740,-85860,0
C00791=40018,59346,-98676,75714,-122693,-85903,0
C00792=40013,59329,-98722,75711,-122679,-85915,0
C00793=39988,59275,-98871,75712,-122628,-85954,0
C00794=39936,59189,-99107,75725,-122539,-86014,0
C00795=39900,59144,-99231,75741,-122487,-86044,0
C00796=39859,59100,-99351,75762,-122433,-86073,0
C00797=39828,59069,-99438,75779,-122394,-86093,0
C00798=39776,58983,-99674,75792,-122306,-86153,0
C00799=30480,51603,-121632,60526,-120465,-93976,0
C00800=30547,51544,-121830,60424,-120409,-94040,0
C00801=30578,51512,-121937,60376,-120376,-94075,0
C00802=30588,51498,-121985,60358,-120360,-94089,0
C00803=30612,51457,-122123,60313,-120313,-94130,0
C00804=30629,51418,-122255,60276,-120265,-94169,0
C00805=30633,51405,-122297,60265,-120250,-94181,0
C00806=30640,51353,-122472,60233,-120181,-94231,0
C00807=30640,51301,-122648,60209,-120110,-94279,0
C00808=30625,51249,-122822,60202,-120033,-94325,0
C00809=30603,51199,-122994,60202,-119956,-94370,0
C00810=30567,51150,-123161,60220,-119875,-94411,0
C00811=30534,51112,-123286,60239,-119812,-94441,0
C00812=30524,51102,-123323,60246,-119794,-94449,0
C00813=30480,51068,-123438,60279,-119732,-94475,0
C00814=30395,51015,-123617,60348,-119629,-94513,0
C00815=30339,50988,-123708,60397,-119573,-94531,0
C00816=30279,50962,-123795,60453,-119518,-94546,0
C00817=30233,50944,-123857,60495,-119477,-94557,0
C00818=30187,50928,-123910,60539,-119440,-94565,0
C00819=30146,50916,-123951,60579,-119409,-94571,0
C00820=30044,50889,-124042,60679,-119338,-94583,0
C00821=29969,50874,-124093,60754,-119292,-94587,0
C00822=29896,50862,-124133,60830,-119251,-94588,0
C00823=29836,50853,-124163,60892,-119218,-94589,0
C00824=29776,50846,-124185,60955,-119189,-94586,0
C00825=29682,50840,-124206,61056,-119149,-94580,0
C00826=29618,50836,-124218,61125,-119123,-94574,0
C00827=29555,50835,-124220,61194,-119101,-94567,0
C00828=29464,50836,-124213,61295,-119073,-94552,0
C00829=29399,50838,-124205,61367,-119055,-94541,0
C00830=29335,50843,-124187,61441,-119040,-94528,0
C00831=29253,50852,-124154,61536,-119025,-94507,0
C00832=29188,50861,-124125,61610,-119016,-94490,0
C00833=29126,50871,-124087,61683,-119009,-94471,0
C00834=29054,50887,-124032,61770,-119007,-94446,0
C00835=28994,50901,-123982,61842,-119005,-94424,0
C00836=28937,50917,-123925,61913,-119009,-94400,0
C00837=28878,50938,-123854,61987,-119017,-94372,0
C00838=28825,50957,-123785,62055,-119026,-94346,0
C00839=28774,50979,-123708,62120,-119039,-94317,0
C00840=28730,51003,-123626,62180,-119056,-94288,0
C00841=28685,51028,-123541,62240,-119074,-94258,0
C00842=28646,51054,-123449,62296,-119096,-94227,0
C00843=28584,51099,-123295,62384,-119135,-94175,0
C00844=28542,51142,-123149,62450,-119178,-94127,0
C00845=28506,51186,-122998,62509,-119224,-94080,0
C00846=28483,51232,-122841,62555,-119277,-94033,0
C00847=28467,51279,-122682,62594,-119333,-93985,0
C00848=28464,51327,-122521,62619,-119395,-93939,0
C00849=28468,51375,-122359,62636,-119459,-93894,0
C00850=28485,51422,-122200,62639,-119527,-93852,0
C00851=28509,51469,-122043,62634,-119596,-93811,0
C00852=28545,51515,-121891,62615,-119667,-93773,0
C00853=28587,51559,-121744,62589,-119740,-93737,0
C00854=28641,51600,-121606,62549,-119812,-93706,0
C00855=28700,51640,-121474,62502,-119885,-93677,0
C00856=28769,51676,-121355,62443,-119956,-93654,0
C00857=28817,51699,-121282,62401,-120002,-93640,0
C00858=28843,51710,-121244,62378,-120026,-93633,0
C00859=28934,51746,-121128,62294,-120104,-93613,0
C00860=28992,51765,-121066,62239,-120150,-93604,0
C00861=29052,51781,-121012,62181,-120192,-93598,0
C00862=29114,51798,-120960,62120,-120236,-93592,0
C00863=29177,51811,-120918,62057,-120275,-93589,0
C00864=29240,51821,-120884,61993,-120311,-93589,0
C00865=29313,51832,-120851,61918,-120351,-93590,0
C00866=29377,51838,-120829,61851,-120383,-93594,0
C00867=29441,51842,-120818,61781,-120412,-93599,0
C00868=29522,51846,-120807,61695,-120445,-93608,0
C00869=29585,51847,-120806,61625,-120469,-93617,0
C00870=29648,51844,-120815,61555,-120489,-93629,0
C00871=29733,51840,-120830,61459,-120514,-93645,0
C00872=29794,51835,-120849,61391,-120528,-93660,0
C00873=29854,51827,-120877,61320,-120540,-93676,0
C00874=29940,51814,-120921,61220,-120553,-93701,0
C00875=29995,51803,-120958,61154,-120559,-93719,0
C00876=30050,51790,-121003,61087,-120561,-93740,0
C00877=30115,51773,-121060,61008,-120563,-93765,0
C00878=30182,51753,-121128,60925,-120559,-93793,0
C00879=30271,51718,-121244,60810,-120545,-93838,0
C00880=30305,51704,-121292,60766,-120538,-93857,0
C00881=30346,51685,-121357,60712,-120527,-93880,0
C00882=30384,51663,-121429,60659,-120512,-93906,0
C00883=30420,51643,-121497,60611,-120497,-93930,0
C00884=30488,51603,-121631,60517,-120468,-93977,0
C00885=25527,55109,-110549,67548,-122413,-90139,0
C00886=36365,52027,-120346,76491,-115352,-91861,0
C00887=36366,51966,-120368,76499,-115372,-91838,0
C00888=25565,55064,-110536,67524,-122464,-90115,0
C00889=36366,51966,-120368,76499,-115372,-91838,0
C00890=39944,50787,-124417,72227,-115645,-93452,0
C00891=35335,53926,-114140,78289,-116451,-89825,0
C00892=36298,54338,-112902,77446,-117220,-89555,0
C00893=40950,51169,-123132,71292,-116424,-93165,0
C00894=40027,50817,-124313,72149,-115708,-93428,0
C00895=35605,54622,-112029,78264,-117082,-89217,0
C00896=36478,55018,-110858,77517,-117802,-88964,0
C00897=42178,51135,-123277,69951,-116843,-93345,0
C00898=33603,54632,-111960,58603,-125571,-91883,0
C00899=34234,54046,-113752,79466,-116000,-89595,0
C00900=35135,54419,-112634,78672,-116704,-89349,0
C00901=34901,54631,-111988,78990,-116734,-89130,0
C00902=35369,54835,-111383,78585,-117110,-88998,0
C00903=35551,54670,-111882,78337,-117089,-89167,0
C00904=36111,54390,-112741,77658,-117166,-89486,0
C00905=34835,54892,-111203,57372,-126390,-91922,0
C00906=36835,53204,-116412,54272,-124993,-93628,0
C00907=39304,53152,-116628,73846,-117667,-91015,0
C00908=44012,55661,-109113,69972,-122078,-89451,0
C00909=34854,54874,-111257,79125,-116876,-88904,0
C00910=33036,56749,-105726,81621,-117061,-87057,0
C00911=36074,53915,-114188,77519,-116798,-89919,0
C00912=40140,51145,-123192,72157,-116096,-93096,0
C00913=40140,51082,-123214,72165,-116118,-93073,0
C00914=25603,55018,-110523,67499,-122515,-90093,0
C00915=36366,51904,-120390,76506,-115390,-91816,0
C00916=36298,54280,-112924,77454,-117236,-89535,0
C00917=40950,51106,-123154,71301,-116447,-93143,0
C00918=39944,50723,-124439,72235,-115668,-93429,0
C00919=35335,53868,-114161,78296,-116467,-89804,0
C00920=36220,54245,-113026,77521,-117172,-89557,0
C00921=35606,54565,-112050,78272,-117098,-89196,0
C00922=36479,54961,-110879,77526,-117819,-88944,0
C00923=42178,51072,-123299,69960,-116867,-93323,0
C00924=33603,54575,-111981,58614,-125598,-91865,0
C00925=34234,53987,-113774,79474,-116016,-89573,0
C00926=35136,54361,-112656,78680,-116721,-89328,0
C00927=34901,54573,-112010,78998,-116750,-89109,0
C00928=35369,54778,-111405,78593,-117127,-88977,0
C00929=35552,54613,-111904,78346,-117105,-89146,0
C00930=36111,54332,-112762,77666,-117183,-89466,0
C00931=41178,50452,-125412,70792,-115813,-93857,0
C00932=36820,53155,-116398,54305,-125034,-93599,0
C00933=39304,53092,-116648,73855,-117687,-90993,0
C00934=43982,55585,-109190,70005,-122068,-89443,0
C00935=34854,54817,-111279,79133,-116891,-88884,0
C00936=33048,56680,-105787,81612,-117074,-87050,0
C00937=36075,53857,-114210,77527,-116815,-89897,0
C00938=40140,51082,-123214,72165,-116118,-93073,0
C00939=40140,51019,-123235,72173,-116141,-93051,0
C00940=25642,54973,-110510,67476,-122567,-90070,0
C00941=36366,51843,-120412,76514,-115410,-91794,0
C00942=36298,54222,-112945,77462,-117253,-89514,0
C00943=40951,51043,-123177,71309,-116470,-93120,0
C00944=39944,50659,-124460,72243,-115690,-93407,0
C00945=35335,53809,-114183,78304,-116484,-89783,0
C00946=36220,54187,-113047,77530,-117190,-89536,0
C00947=35606,54507,-112071,78281,-117114,-89175,0
C00948=36479,54904,-110901,77534,-117836,-88923,0
C00949=42179,51009,-123320,69968,-116891,-93300,0
C00950=33603,54517,-112002,58626,-125626,-91847,0
C00951=34235,53929,-113795,79481,-116033,-89553,0
C00952=35136,54303,-112677,78688,-116737,-89307,0
C00953=34901,54516,-112031,79006,-116766,-89088,0
C00954=35369,54721,-111426,78602,-117144,-88956,0
C00955=35552,54555,-111925,78354,-117121,-89125,0
C00956=36112,54274,-112784,77674,-117199,-89445,0
C00957=41179,50387,-125434,70800,-115837,-93834,0
C00958=36806,53107,-116384,54338,-125074,-93569,0
C00959=39304,53033,-116670,73863,-117707,-90972,0
C00960=43952,55510,-109267,70039,-122056,-89435,0
C00961=34855,54759,-111300,79141,-116907,-88863,0
C00962=33060,56611,-105848,81603,-117086,-87043,0
C00963=36075,53798,-114231,77535,-116832,-89876,0
C00964=40140,51019,-123235,72173,-116141,-93051,0
C00965=40141,50956,-123257,72181,-116164,-93028,0
C00966=25680,54928,-110497,67452,-122618,-90046,0
C00967=36367,51781,-120434,76522,-115428,-91771,0
C00968=36298,54164,-112966,77471,-117270,-89493,0
C00969=40951,50979,-123199,71317,-116493,-93098,0
C00970=39945,50595,-124482,72251,-115713,-93384,0
C00971=35336,53750,-114204,78312,-116500,-89762,0
C00972=36221,54129,-113069,77538,-117207,-89515,0
C00973=35606,54449,-112092,78289,-117130,-89154,0
C00974=36479,54847,-110922,77543,-117853,-88903,0
C00975=42179,50946,-123342,69976,-116915,-93278,0
C00976=33603,54459,-112023,58637,-125653,-91829,0
C00977=34235,53870,-113816,79489,-116049,-89531,0
C00978=35137,54245,-112698,78696,-116753,-89286,0
C00979=34902,54458,-112052,79014,-116782,-89067,0
C00980=35370,54663,-111447,78610,-117160,-88935,0
C00981=35552,54498,-111946,78362,-117137,-89105,0
C00982=36112,54216,-112805,77682,-117216,-89424,0
C00983=41179,50323,-125456,70808,-115861,-93812,0
C00984=36792,53059,-116370,54371,-125115,-93540,0
//INST
///DATE 2025/02/20 16:20
///COMM Generated using RoboDK
///ATTR SC,RW
///GROUP1 RB1
NOP
MOVL C00000 V=30.0 PL=1
MOVL C00001 V=30.0 PL=1
MOVL C00002 V=30.0 PL=1
MOVL C00003 V=30.0 PL=1
MOVL C00004 V=30.0 PL=1
MOVL C00005 V=30.0 PL=1
MOVL C00006 V=30.0 PL=1
MOVL C00007 V=30.0 PL=1
MOVL C00008 V=30.0 PL=1
MOVL C00009 V=30.0 PL=1
MOVL C00010 V=30.0 PL=1
MOVL C00011 V=30.0 PL=1
MOVL C00012 V=130.0 PL=1
MOVL C00013 V=130.0 PL=1
MOVL C00014 V=30.0 PL=1
MOVL C00015 V=30.0 PL=1
MOVL C00016 V=30.0 PL=1
MOVL C00017 V=30.0 PL=1
MOVL C00018 V=30.0 PL=1
MOVL C00019 V=30.0 PL=1
MOVL C00020 V=30.0 PL=1
MOVL C00021 V=30.0 PL=1
MOVL C00022 V=30.0 PL=1
MOVL C00023 V=30.0 PL=1
MOVL C00024 V=30.0 PL=1
MOVL C00025 V=30.0 PL=1
MOVL C00026 V=30.0 PL=1
MOVL C00027 V=30.0 PL=1
MOVL C00028 V=30.0 PL=1
MOVL C00029 V=30.0 PL=1
MOVL C00030 V=30.0 PL=1
MOVL C00031 V=30.0 PL=1
MOVL C00032 V=30.0 PL=1
MOVL C00033 V=30.0 PL=1
MOVL C00034 V=30.0 PL=1
MOVL C00035 V=30.0 PL=1
MOVL C00036 V=30.0 PL=1
MOVL C00037 V=30.0 PL=1
MOVL C00038 V=30.0 PL=1
MOVL C00039 V=30.0 PL=1
MOVL C00040 V=30.0 PL=1
MOVL C00041 V=30.0 PL=1
MOVL C00042 V=30.0 PL=1
MOVL C00043 V=30.0 PL=1
MOVL C00044 V=30.0 PL=1
MOVL C00045 V=30.0 PL=1
MOVL C00046 V=30.0 PL=1
MOVL C00047 V=30.0 PL=1
MOVL C00048 V=30.0 PL=1
MOVL C00049 V=30.0 PL=1
MOVL C00050 V=30.0 PL=1
MOVL C00051 V=30.0 PL=1
MOVL C00052 V=30.0 PL=1
MOVL C00053 V=30.0 PL=1
MOVL C00054 V=30.0 PL=1
MOVL C00055 V=30.0 PL=1
MOVL C00056 V=30.0 PL=1
MOVL C00057 V=30.0 PL=1
MOVL C00058 V=30.0 PL=1
MOVL C00059 V=30.0 PL=1
MOVL C00060 V=30.0 PL=1
MOVL C00061 V=30.0 PL=1
MOVL C00062 V=30.0 PL=1
MOVL C00063 V=30.0 PL=1
MOVL C00064 V=30.0 PL=1
MOVL C00065 V=30.0 PL=1
MOVL C00066 V=30.0 PL=1
MOVL C00067 V=30.0 PL=1
MOVL C00068 V=30.0 PL=1
MOVL C00069 V=30.0 PL=1
MOVL C00070 V=30.0 PL=1
MOVL C00071 V=30.0 PL=1
MOVL C00072 V=30.0 PL=1
MOVL C00073 V=30.0 PL=1
MOVL C00074 V=30.0 PL=1
MOVL C00075 V=30.0 PL=1
MOVL C00076 V=30.0 PL=1
MOVL C00077 V=30.0 PL=1
MOVL C00078 V=30.0 PL=1
MOVL C00079 V=30.0 PL=1
MOVL C00080 V=30.0 PL=1
MOVL C00081 V=30.0 PL=1
MOVL C00082 V=30.0 PL=1
MOVL C00083 V=30.0 PL=1
MOVL C00084 V=30.0 PL=1
MOVL C00085 V=30.0 PL=1
MOVL C00086 V=30.0 PL=1
MOVL C00087 V=30.0 PL=1
MOVL C00088 V=130.0 PL=1
MOVL C00089 V=130.0 PL=1
MOVL C00090 V=30.0 PL=1
MOVL C00091 V=130.0 PL=1
MOVL C00092 V=30.0 PL=1
MOVL C00093 V=30.0 PL=1
MOVL C00094 V=30.0 PL=1
MOVL C00095 V=30.0 PL=1
MOVL C00096 V=30.0 PL=1
MOVL C00097 V=30.0 PL=1
MOVL C00098 V=30.0 PL=1
MOVL C00099 V=30.0 PL=1
MOVL C00100 V=30.0 PL=1
MOVL C00101 V=30.0 PL=1
MOVL C00102 V=30.0 PL=1
MOVL C00103 V=30.0 PL=1
MOVL C00104 V=30.0 PL=1
MOVL C00105 V=30.0 PL=1
MOVL C00106 V=30.0 PL=1
MOVL C00107 V=30.0 PL=1
MOVL C00108 V=30.0 PL=1
MOVL C00109 V=30.0 PL=1
MOVL C00110 V=30.0 PL=1
MOVL C00111 V=30.0 PL=1
MOVL C00112 V=30.0 PL=1
MOVL C00113 V=30.0 PL=1
MOVL C00114 V=30.0 PL=1
MOVL C00115 V=30.0 PL=1
MOVL C00116 V=30.0 PL=1
MOVL C00117 V=30.0 PL=1
MOVL C00118 V=30.0 PL=1
MOVL C00119 V=30.0 PL=1
MOVL C00120 V=30.0 PL=1
MOVL C00121 V=30.0 PL=1
MOVL C00122 V=30.0 PL=1
MOVL C00123 V=30.0 PL=1
MOVL C00124 V=30.0 PL=1
MOVL C00125 V=30.0 PL=1
MOVL C00126 V=30.0 PL=1
MOVL C00127 V=30.0 PL=1
MOVL C00128 V=30.0 PL=1
MOVL C00129 V=30.0 PL=1
MOVL C00130 V=30.0 PL=1
MOVL C00131 V=30.0 PL=1
MOVL C00132 V=30.0 PL=1
MOVL C00133 V=30.0 PL=1
MOVL C00134 V=30.0 PL=1
MOVL C00135 V=30.0 PL=1
MOVL C00136 V=30.0 PL=1
MOVL C00137 V=30.0 PL=1
MOVL C00138 V=30.0 PL=1
MOVL C00139 V=30.0 PL=1
MOVL C00140 V=30.0 PL=1
MOVL C00141 V=30.0 PL=1
MOVL C00142 V=30.0 PL=1
MOVL C00143 V=30.0 PL=1
MOVL C00144 V=30.0 PL=1
MOVL C00145 V=30.0 PL=1
MOVL C00146 V=30.0 PL=1
MOVL C00147 V=30.0 PL=1
MOVL C00148 V=30.0 PL=1
MOVL C00149 V=30.0 PL=1
MOVL C00150 V=30.0 PL=1
MOVL C00151 V=30.0 PL=1
MOVL C00152 V=30.0 PL=1
MOVL C00153 V=30.0 PL=1
MOVL C00154 V=30.0 PL=1
MOVL C00155 V=30.0 PL=1
MOVL C00156 V=30.0 PL=1
MOVL C00157 V=30.0 PL=1
MOVL C00158 V=30.0 PL=1
MOVL C00159 V=30.0 PL=1
MOVL C00160 V=30.0 PL=1
MOVL C00161 V=30.0 PL=1
MOVL C00162 V=30.0 PL=1
MOVL C00163 V=30.0 PL=1
MOVL C00164 V=30.0 PL=1
MOVL C00165 V=130.0 PL=1
MOVL C00166 V=130.0 PL=1
MOVL C00167 V=130.0 PL=1
MOVL C00168 V=30.0 PL=1
MOVL C00169 V=30.0 PL=1
MOVL C00170 V=30.0 PL=1
MOVL C00171 V=30.0 PL=1
MOVL C00172 V=30.0 PL=1
MOVL C00173 V=30.0 PL=1
MOVL C00174 V=30.0 PL=1
MOVL C00175 V=30.0 PL=1
MOVL C00176 V=30.0 PL=1
MOVL C00177 V=30.0 PL=1
MOVL C00178 V=30.0 PL=1
MOVL C00179 V=30.0 PL=1
MOVL C00180 V=30.0 PL=1
MOVL C00181 V=30.0 PL=1
MOVL C00182 V=30.0 PL=1
MOVL C00183 V=30.0 PL=1
MOVL C00184 V=30.0 PL=1
MOVL C00185 V=30.0 PL=1
MOVL C00186 V=30.0 PL=1
MOVL C00187 V=30.0 PL=1
MOVL C00188 V=30.0 PL=1
MOVL C00189 V=30.0 PL=1
MOVL C00190 V=30.0 PL=1
MOVL C00191 V=30.0 PL=1
MOVL C00192 V=30.0 PL=1
MOVL C00193 V=30.0 PL=1
MOVL C00194 V=30.0 PL=1
MOVL C00195 V=30.0 PL=1
MOVL C00196 V=30.0 PL=1
MOVL C00197 V=30.0 PL=1
MOVL C00198 V=30.0 PL=1
MOVL C00199 V=30.0 PL=1
MOVL C00200 V=30.0 PL=1
MOVL C00201 V=30.0 PL=1
MOVL C00202 V=30.0 PL=1
MOVL C00203 V=30.0 PL=1
MOVL C00204 V=30.0 PL=1
MOVL C00205 V=30.0 PL=1
MOVL C00206 V=30.0 PL=1
MOVL C00207 V=30.0 PL=1
MOVL C00208 V=30.0 PL=1
MOVL C00209 V=30.0 PL=1
MOVL C00210 V=30.0 PL=1
MOVL C00211 V=30.0 PL=1
MOVL C00212 V=30.0 PL=1
MOVL C00213 V=30.0 PL=1
MOVL C00214 V=30.0 PL=1
MOVL C00215 V=30.0 PL=1
MOVL C00216 V=30.0 PL=1
MOVL C00217 V=30.0 PL=1
MOVL C00218 V=30.0 PL=1
MOVL C00219 V=30.0 PL=1
MOVL C00220 V=30.0 PL=1
MOVL C00221 V=30.0 PL=1
MOVL C00222 V=30.0 PL=1
MOVL C00223 V=30.0 PL=1
MOVL C00224 V=30.0 PL=1
MOVL C00225 V=30.0 PL=1
MOVL C00226 V=30.0 PL=1
MOVL C00227 V=30.0 PL=1
MOVL C00228 V=30.0 PL=1
MOVL C00229 V=30.0 PL=1
MOVL C00230 V=30.0 PL=1
MOVL C00231 V=30.0 PL=1
MOVL C00232 V=30.0 PL=1
MOVL C00233 V=30.0 PL=1
MOVL C00234 V=30.0 PL=1
MOVL C00235 V=30.0 PL=1
MOVL C00236 V=30.0 PL=1
MOVL C00237 V=30.0 PL=1
MOVL C00238 V=30.0 PL=1
MOVL C00239 V=30.0 PL=1
MOVL C00240 V=30.0 PL=1
MOVL C00241 V=30.0 PL=1
MOVL C00242 V=30.0 PL=1
MOVL C00243 V=30.0 PL=1
MOVL C00244 V=30.0 PL=1
MOVL C00245 V=30.0 PL=1
MOVL C00246 V=30.0 PL=1
MOVL C00247 V=30.0 PL=1
MOVL C00248 V=30.0 PL=1
MOVL C00249 V=30.0 PL=1
MOVL C00250 V=30.0 PL=1
MOVL C00251 V=30.0 PL=1
MOVL C00252 V=30.0 PL=1
MOVL C00253 V=30.0 PL=1
MOVL C00254 V=130.0 PL=1
MOVL C00255 V=130.0 PL=1
MOVL C00256 V=60.0 PL=1
MOVL C00257 V=60.0 PL=1
MOVL C00258 V=60.0 PL=1
MOVL C00259 V=60.0 PL=1
MOVL C00260 V=130.0 PL=1
MOVL C00261 V=30.0 PL=1
MOVL C00262 V=30.0 PL=1
MOVL C00263 V=30.0 PL=1
MOVL C00264 V=30.0 PL=1
MOVL C00265 V=30.0 PL=1
MOVL C00266 V=30.0 PL=1
MOVL C00267 V=30.0 PL=1
MOVL C00268 V=30.0 PL=1
MOVL C00269 V=130.0 PL=1
MOVL C00270 V=130.0 PL=1
MOVL C00271 V=30.0 PL=1
MOVL C00272 V=130.0 PL=1
MOVL C00273 V=30.0 PL=1
MOVL C00274 V=130.0 PL=1
MOVL C00275 V=30.0 PL=1
MOVL C00276 V=130.0 PL=1
MOVL C00277 V=20.0 PL=1
MOVL C00278 V=130.0 PL=1
MOVL C00279 V=30.0 PL=1
MOVL C00280 V=30.0 PL=1
MOVL C00281 V=30.0 PL=1
MOVL C00282 V=30.0 PL=1
MOVL C00283 V=30.0 PL=1
MOVL C00284 V=30.0 PL=1
MOVL C00285 V=30.0 PL=1
MOVL C00286 V=30.0 PL=1
MOVL C00287 V=30.0 PL=1
MOVL C00288 V=30.0 PL=1
MOVL C00289 V=30.0 PL=1
MOVL C00290 V=30.0 PL=1
MOVL C00291 V=30.0 PL=1
MOVL C00292 V=30.0 PL=1
MOVL C00293 V=30.0 PL=1
MOVL C00294 V=30.0 PL=1
MOVL C00295 V=30.0 PL=1
MOVL C00296 V=30.0 PL=1
MOVL C00297 V=30.0 PL=1
MOVL C00298 V=30.0 PL=1
MOVL C00299 V=30.0 PL=1
MOVL C00300 V=30.0 PL=1
MOVL C00301 V=30.0 PL=1
MOVL C00302 V=30.0 PL=1
MOVL C00303 V=30.0 PL=1
MOVL C00304 V=30.0 PL=1
MOVL C00305 V=30.0 PL=1
MOVL C00306 V=30.0 PL=1
MOVL C00307 V=30.0 PL=1
MOVL C00308 V=30.0 PL=1
MOVL C00309 V=30.0 PL=1
MOVL C00310 V=30.0 PL=1
MOVL C00311 V=30.0 PL=1
MOVL C00312 V=30.0 PL=1
MOVL C00313 V=30.0 PL=1
MOVL C00314 V=30.0 PL=1
MOVL C00315 V=30.0 PL=1
MOVL C00316 V=30.0 PL=1
MOVL C00317 V=30.0 PL=1
MOVL C00318 V=30.0 PL=1
MOVL C00319 V=30.0 PL=1
MOVL C00320 V=30.0 PL=1
MOVL C00321 V=30.0 PL=1
MOVL C00322 V=30.0 PL=1
MOVL C00323 V=30.0 PL=1
MOVL C00324 V=30.0 PL=1
MOVL C00325 V=30.0 PL=1
MOVL C00326 V=30.0 PL=1
MOVL C00327 V=30.0 PL=1
MOVL C00328 V=30.0 PL=1
MOVL C00329 V=30.0 PL=1
MOVL C00330 V=30.0 PL=1
MOVL C00331 V=30.0 PL=1
MOVL C00332 V=30.0 PL=1
MOVL C00333 V=30.0 PL=1
MOVL C00334 V=30.0 PL=1
MOVL C00335 V=30.0 PL=1
MOVL C00336 V=30.0 PL=1
MOVL C00337 V=30.0 PL=1
MOVL C00338 V=30.0 PL=1
MOVL C00339 V=30.0 PL=1
MOVL C00340 V=30.0 PL=1
MOVL C00341 V=30.0 PL=1
MOVL C00342 V=30.0 PL=1
MOVL C00343 V=30.0 PL=1
MOVL C00344 V=30.0 PL=1
MOVL C00345 V=30.0 PL=1
MOVL C00346 V=30.0 PL=1
MOVL C00347 V=30.0 PL=1
MOVL C00348 V=30.0 PL=1
MOVL C00349 V=30.0 PL=1
MOVL C00350 V=30.0 PL=1
MOVL C00351 V=30.0 PL=1
MOVL C00352 V=30.0 PL=1
MOVL C00353 V=30.0 PL=1
MOVL C00354 V=30.0 PL=1
MOVL C00355 V=30.0 PL=1
MOVL C00356 V=30.0 PL=1
MOVL C00357 V=30.0 PL=1
MOVL C00358 V=30.0 PL=1
MOVL C00359 V=30.0 PL=1
MOVL C00360 V=30.0 PL=1
MOVL C00361 V=30.0 PL=1
MOVL C00362 V=30.0 PL=1
MOVL C00363 V=30.0 PL=1
MOVL C00364 V=130.0 PL=1
MOVL C00365 V=130.0 PL=1
MOVL C00366 V=30.0 PL=1
MOVL C00367 V=30.0 PL=1
MOVL C00368 V=30.0 PL=1
MOVL C00369 V=30.0 PL=1
MOVL C00370 V=30.0 PL=1
MOVL C00371 V=30.0 PL=1
MOVL C00372 V=30.0 PL=1
MOVL C00373 V=30.0 PL=1
MOVL C00374 V=30.0 PL=1
MOVL C00375 V=30.0 PL=1
MOVL C00376 V=30.0 PL=1
MOVL C00377 V=30.0 PL=1
MOVL C00378 V=30.0 PL=1
MOVL C00379 V=30.0 PL=1
MOVL C00380 V=30.0 PL=1
MOVL C00381 V=30.0 PL=1
MOVL C00382 V=30.0 PL=1
MOVL C00383 V=30.0 PL=1
MOVL C00384 V=30.0 PL=1
MOVL C00385 V=30.0 PL=1
MOVL C00386 V=30.0 PL=1
MOVL C00387 V=30.0 PL=1
MOVL C00388 V=30.0 PL=1
MOVL C00389 V=30.0 PL=1
MOVL C00390 V=30.0 PL=1
MOVL C00391 V=30.0 PL=1
MOVL C00392 V=30.0 PL=1
MOVL C00393 V=30.0 PL=1
MOVL C00394 V=30.0 PL=1
MOVL C00395 V=30.0 PL=1
MOVL C00396 V=30.0 PL=1
MOVL C00397 V=30.0 PL=1
MOVL C00398 V=30.0 PL=1
MOVL C00399 V=30.0 PL=1
MOVL C00400 V=30.0 PL=1
MOVL C00401 V=30.0 PL=1
MOVL C00402 V=30.0 PL=1
MOVL C00403 V=30.0 PL=1
MOVL C00404 V=30.0 PL=1
MOVL C00405 V=30.0 PL=1
MOVL C00406 V=30.0 PL=1
MOVL C00407 V=30.0 PL=1
MOVL C00408 V=30.0 PL=1
MOVL C00409 V=30.0 PL=1
MOVL C00410 V=30.0 PL=1
MOVL C00411 V=30.0 PL=1
MOVL C00412 V=30.0 PL=1
MOVL C00413 V=30.0 PL=1
MOVL C00414 V=30.0 PL=1
MOVL C00415 V=30.0 PL=1
MOVL C00416 V=30.0 PL=1
MOVL C00417 V=30.0 PL=1
MOVL C00418 V=30.0 PL=1
MOVL C00419 V=30.0 PL=1
MOVL C00420 V=30.0 PL=1
MOVL C00421 V=30.0 PL=1
MOVL C00422 V=30.0 PL=1
MOVL C00423 V=30.0 PL=1
MOVL C00424 V=30.0 PL=1
MOVL C00425 V=30.0 PL=1
MOVL C00426 V=30.0 PL=1
MOVL C00427 V=30.0 PL=1
MOVL C00428 V=30.0 PL=1
MOVL C00429 V=30.0 PL=1
MOVL C00430 V=30.0 PL=1
MOVL C00431 V=30.0 PL=1
MOVL C00432 V=30.0 PL=1
MOVL C00433 V=30.0 PL=1
MOVL C00434 V=30.0 PL=1
MOVL C00435 V=30.0 PL=1
MOVL C00436 V=30.0 PL=1
MOVL C00437 V=30.0 PL=1
MOVL C00438 V=30.0 PL=1
MOVL C00439 V=30.0 PL=1
MOVL C00440 V=30.0 PL=1
MOVL C00441 V=30.0 PL=1
MOVL C00442 V=30.0 PL=1
MOVL C00443 V=30.0 PL=1
MOVL C00444 V=30.0 PL=1
MOVL C00445 V=30.0 PL=1
MOVL C00446 V=30.0 PL=1
MOVL C00447 V=30.0 PL=1
MOVL C00448 V=30.0 PL=1
MOVL C00449 V=30.0 PL=1
MOVL C00450 V=30.0 PL=1
MOVL C00451 V=130.0 PL=1
MOVL C00452 V=130.0 PL=1
MOVL C00453 V=30.0 PL=1
MOVL C00454 V=30.0 PL=1
MOVL C00455 V=30.0 PL=1
MOVL C00456 V=30.0 PL=1
MOVL C00457 V=30.0 PL=1
MOVL C00458 V=30.0 PL=1
MOVL C00459 V=30.0 PL=1
MOVL C00460 V=30.0 PL=1
MOVL C00461 V=30.0 PL=1
MOVL C00462 V=30.0 PL=1
MOVL C00463 V=30.0 PL=1
MOVL C00464 V=30.0 PL=1
MOVL C00465 V=30.0 PL=1
MOVL C00466 V=30.0 PL=1
MOVL C00467 V=30.0 PL=1
MOVL C00468 V=30.0 PL=1
MOVL C00469 V=30.0 PL=1
MOVL C00470 V=30.0 PL=1
MOVL C00471 V=30.0 PL=1
MOVL C00472 V=30.0 PL=1
MOVL C00473 V=30.0 PL=1
MOVL C00474 V=30.0 PL=1
MOVL C00475 V=30.0 PL=1
MOVL C00476 V=30.0 PL=1
MOVL C00477 V=30.0 PL=1
MOVL C00478 V=30.0 PL=1
MOVL C00479 V=30.0 PL=1
MOVL C00480 V=30.0 PL=1
MOVL C00481 V=30.0 PL=1
MOVL C00482 V=30.0 PL=1
MOVL C00483 V=30.0 PL=1
MOVL C00484 V=30.0 PL=1
MOVL C00485 V=30.0 PL=1
MOVL C00486 V=30.0 PL=1
MOVL C00487 V=30.0 PL=1
MOVL C00488 V=30.0 PL=1
MOVL C00489 V=30.0 PL=1
MOVL C00490 V=30.0 PL=1
MOVL C00491 V=30.0 PL=1
MOVL C00492 V=30.0 PL=1
MOVL C00493 V=30.0 PL=1
MOVL C00494 V=30.0 PL=1
MOVL C00495 V=30.0 PL=1
MOVL C00496 V=30.0 PL=1
MOVL C00497 V=30.0 PL=1
MOVL C00498 V=30.0 PL=1
MOVL C00499 V=30.0 PL=1
MOVL C00500 V=30.0 PL=1
MOVL C00501 V=30.0 PL=1
MOVL C00502 V=30.0 PL=1
MOVL C00503 V=30.0 PL=1
MOVL C00504 V=30.0 PL=1
MOVL C00505 V=30.0 PL=1
MOVL C00506 V=30.0 PL=1
MOVL C00507 V=30.0 PL=1
MOVL C00508 V=30.0 PL=1
MOVL C00509 V=30.0 PL=1
MOVL C00510 V=30.0 PL=1
MOVL C00511 V=30.0 PL=1
MOVL C00512 V=30.0 PL=1
MOVL C00513 V=30.0 PL=1
MOVL C00514 V=30.0 PL=1
MOVL C00515 V=30.0 PL=1
MOVL C00516 V=30.0 PL=1
MOVL C00517 V=30.0 PL=1
MOVL C00518 V=30.0 PL=1
MOVL C00519 V=30.0 PL=1
MOVL C00520 V=30.0 PL=1
MOVL C00521 V=30.0 PL=1
MOVL C00522 V=30.0 PL=1
MOVL C00523 V=30.0 PL=1
MOVL C00524 V=30.0 PL=1
MOVL C00525 V=30.0 PL=1
MOVL C00526 V=30.0 PL=1
MOVL C00527 V=30.0 PL=1
MOVL C00528 V=130.0 PL=1
MOVL C00529 V=130.0 PL=1
MOVL C00530 V=30.0 PL=1
MOVL C00531 V=130.0 PL=1
MOVL C00532 V=130.0 PL=1
MOVL C00533 V=30.0 PL=1
MOVL C00534 V=30.0 PL=1
MOVL C00535 V=30.0 PL=1
MOVL C00536 V=30.0 PL=1
MOVL C00537 V=30.0 PL=1
MOVL C00538 V=30.0 PL=1
MOVL C00539 V=30.0 PL=1
MOVL C00540 V=30.0 PL=1
MOVL C00541 V=30.0 PL=1
MOVL C00542 V=30.0 PL=1
MOVL C00543 V=30.0 PL=1
MOVL C00544 V=30.0 PL=1
MOVL C00545 V=30.0 PL=1
MOVL C00546 V=30.0 PL=1
MOVL C00547 V=30.0 PL=1
MOVL C00548 V=30.0 PL=1
MOVL C00549 V=30.0 PL=1
MOVL C00550 V=30.0 PL=1
MOVL C00551 V=30.0 PL=1
MOVL C00552 V=30.0 PL=1
MOVL C00553 V=30.0 PL=1
MOVL C00554 V=30.0 PL=1
MOVL C00555 V=30.0 PL=1
MOVL C00556 V=30.0 PL=1
MOVL C00557 V=30.0 PL=1
MOVL C00558 V=30.0 PL=1
MOVL C00559 V=30.0 PL=1
MOVL C00560 V=30.0 PL=1
MOVL C00561 V=30.0 PL=1
MOVL C00562 V=30.0 PL=1
MOVL C00563 V=30.0 PL=1
MOVL C00564 V=30.0 PL=1
MOVL C00565 V=30.0 PL=1
MOVL C00566 V=30.0 PL=1
MOVL C00567 V=30.0 PL=1
MOVL C00568 V=30.0 PL=1
MOVL C00569 V=30.0 PL=1
MOVL C00570 V=30.0 PL=1
MOVL C00571 V=30.0 PL=1
MOVL C00572 V=30.0 PL=1
MOVL C00573 V=30.0 PL=1
MOVL C00574 V=30.0 PL=1
MOVL C00575 V=30.0 PL=1
MOVL C00576 V=30.0 PL=1
MOVL C00577 V=30.0 PL=1
MOVL C00578 V=30.0 PL=1
MOVL C00579 V=30.0 PL=1
MOVL C00580 V=30.0 PL=1
MOVL C00581 V=30.0 PL=1
MOVL C00582 V=30.0 PL=1
MOVL C00583 V=30.0 PL=1
MOVL C00584 V=30.0 PL=1
MOVL C00585 V=30.0 PL=1
MOVL C00586 V=30.0 PL=1
MOVL C00587 V=30.0 PL=1
MOVL C00588 V=30.0 PL=1
MOVL C00589 V=30.0 PL=1
MOVL C00590 V=30.0 PL=1
MOVL C00591 V=30.0 PL=1
MOVL C00592 V=30.0 PL=1
MOVL C00593 V=30.0 PL=1
MOVL C00594 V=30.0 PL=1
MOVL C00595 V=30.0 PL=1
MOVL C00596 V=30.0 PL=1
MOVL C00597 V=30.0 PL=1
MOVL C00598 V=30.0 PL=1
MOVL C00599 V=30.0 PL=1
MOVL C00600 V=30.0 PL=1
MOVL C00601 V=30.0 PL=1
MOVL C00602 V=30.0 PL=1
MOVL C00603 V=30.0 PL=1
MOVL C00604 V=30.0 PL=1
MOVL C00605 V=30.0 PL=1
MOVL C00606 V=30.0 PL=1
MOVL C00607 V=30.0 PL=1
MOVL C00608 V=30.0 PL=1
MOVL C00609 V=30.0 PL=1
MOVL C00610 V=130.0 PL=1
MOVL C00611 V=130.0 PL=1
MOVL C00612 V=60.0 PL=1
MOVL C00613 V=60.0 PL=1
MOVL C00614 V=60.0 PL=1
MOVL C00615 V=60.0 PL=1
MOVL C00616 V=130.0 PL=1
MOVL C00617 V=30.0 PL=1
MOVL C00618 V=30.0 PL=1
MOVL C00619 V=30.0 PL=1
MOVL C00620 V=30.0 PL=1
MOVL C00621 V=30.0 PL=1
MOVL C00622 V=30.0 PL=1
MOVL C00623 V=30.0 PL=1
MOVL C00624 V=30.0 PL=1
MOVL C00625 V=130.0 PL=1
MOVL C00626 V=130.0 PL=1
MOVL C00627 V=30.0 PL=1
MOVL C00628 V=130.0 PL=1
MOVL C00629 V=30.0 PL=1
MOVL C00630 V=130.0 PL=1
MOVL C00631 V=30.0 PL=1
MOVL C00632 V=130.0 PL=1
MOVL C00633 V=20.0 PL=1
MOVL C00634 V=130.0 PL=1
MOVL C00635 V=30.0 PL=1
MOVL C00636 V=30.0 PL=1
MOVL C00637 V=30.0 PL=1
MOVL C00638 V=30.0 PL=1
MOVL C00639 V=30.0 PL=1
MOVL C00640 V=30.0 PL=1
MOVL C00641 V=30.0 PL=1
MOVL C00642 V=30.0 PL=1
MOVL C00643 V=30.0 PL=1
MOVL C00644 V=30.0 PL=1
MOVL C00645 V=30.0 PL=1
MOVL C00646 V=30.0 PL=1
MOVL C00647 V=30.0 PL=1
MOVL C00648 V=30.0 PL=1
MOVL C00649 V=30.0 PL=1
MOVL C00650 V=30.0 PL=1
MOVL C00651 V=30.0 PL=1
MOVL C00652 V=30.0 PL=1
MOVL C00653 V=30.0 PL=1
MOVL C00654 V=30.0 PL=1
MOVL C00655 V=30.0 PL=1
MOVL C00656 V=30.0 PL=1
MOVL C00657 V=30.0 PL=1
MOVL C00658 V=30.0 PL=1
MOVL C00659 V=30.0 PL=1
MOVL C00660 V=30.0 PL=1
MOVL C00661 V=30.0 PL=1
MOVL C00662 V=30.0 PL=1
MOVL C00663 V=30.0 PL=1
MOVL C00664 V=30.0 PL=1
MOVL C00665 V=30.0 PL=1
MOVL C00666 V=30.0 PL=1
MOVL C00667 V=30.0 PL=1
MOVL C00668 V=30.0 PL=1
MOVL C00669 V=30.0 PL=1
MOVL C00670 V=30.0 PL=1
MOVL C00671 V=30.0 PL=1
MOVL C00672 V=30.0 PL=1
MOVL C00673 V=30.0 PL=1
MOVL C00674 V=30.0 PL=1
MOVL C00675 V=30.0 PL=1
MOVL C00676 V=30.0 PL=1
MOVL C00677 V=30.0 PL=1
MOVL C00678 V=30.0 PL=1
MOVL C00679 V=30.0 PL=1
MOVL C00680 V=30.0 PL=1
MOVL C00681 V=30.0 PL=1
MOVL C00682 V=30.0 PL=1
MOVL C00683 V=30.0 PL=1
MOVL C00684 V=30.0 PL=1
MOVL C00685 V=30.0 PL=1
MOVL C00686 V=30.0 PL=1
MOVL C00687 V=30.0 PL=1
MOVL C00688 V=30.0 PL=1
MOVL C00689 V=30.0 PL=1
MOVL C00690 V=30.0 PL=1
MOVL C00691 V=30.0 PL=1
MOVL C00692 V=30.0 PL=1
MOVL C00693 V=30.0 PL=1
MOVL C00694 V=30.0 PL=1
MOVL C00695 V=30.0 PL=1
MOVL C00696 V=30.0 PL=1
MOVL C00697 V=30.0 PL=1
MOVL C00698 V=30.0 PL=1
MOVL C00699 V=30.0 PL=1
MOVL C00700 V=30.0 PL=1
MOVL C00701 V=30.0 PL=1
MOVL C00702 V=30.0 PL=1
MOVL C00703 V=30.0 PL=1
MOVL C00704 V=30.0 PL=1
MOVL C00705 V=30.0 PL=1
MOVL C00706 V=30.0 PL=1
MOVL C00707 V=30.0 PL=1
MOVL C00708 V=30.0 PL=1
MOVL C00709 V=30.0 PL=1
MOVL C00710 V=30.0 PL=1
MOVL C00711 V=30.0 PL=1
MOVL C00712 V=30.0 PL=1
MOVL C00713 V=130.0 PL=1
MOVL C00714 V=130.0 PL=1
MOVL C00715 V=30.0 PL=1
MOVL C00716 V=30.0 PL=1
MOVL C00717 V=30.0 PL=1
MOVL C00718 V=30.0 PL=1
MOVL C00719 V=30.0 PL=1
MOVL C00720 V=30.0 PL=1
MOVL C00721 V=30.0 PL=1
MOVL C00722 V=30.0 PL=1
MOVL C00723 V=30.0 PL=1
MOVL C00724 V=30.0 PL=1
MOVL C00725 V=30.0 PL=1
MOVL C00726 V=30.0 PL=1
MOVL C00727 V=30.0 PL=1
MOVL C00728 V=30.0 PL=1
MOVL C00729 V=30.0 PL=1
MOVL C00730 V=30.0 PL=1
MOVL C00731 V=30.0 PL=1
MOVL C00732 V=30.0 PL=1
MOVL C00733 V=30.0 PL=1
MOVL C00734 V=30.0 PL=1
MOVL C00735 V=30.0 PL=1
MOVL C00736 V=30.0 PL=1
MOVL C00737 V=30.0 PL=1
MOVL C00738 V=30.0 PL=1
MOVL C00739 V=30.0 PL=1
MOVL C00740 V=30.0 PL=1
MOVL C00741 V=30.0 PL=1
MOVL C00742 V=30.0 PL=1
MOVL C00743 V=30.0 PL=1
MOVL C00744 V=30.0 PL=1
MOVL C00745 V=30.0 PL=1
MOVL C00746 V=30.0 PL=1
MOVL C00747 V=30.0 PL=1
MOVL C00748 V=30.0 PL=1
MOVL C00749 V=30.0 PL=1
MOVL C00750 V=30.0 PL=1
MOVL C00751 V=30.0 PL=1
MOVL C00752 V=30.0 PL=1
MOVL C00753 V=30.0 PL=1
MOVL C00754 V=30.0 PL=1
MOVL C00755 V=30.0 PL=1
MOVL C00756 V=30.0 PL=1
MOVL C00757 V=30.0 PL=1
MOVL C00758 V=30.0 PL=1
MOVL C00759 V=30.0 PL=1
MOVL C00760 V=30.0 PL=1
MOVL C00761 V=30.0 PL=1
MOVL C00762 V=30.0 PL=1
MOVL C00763 V=30.0 PL=1
MOVL C00764 V=30.0 PL=1
MOVL C00765 V=30.0 PL=1
MOVL C00766 V=30.0 PL=1
MOVL C00767 V=30.0 PL=1
MOVL C00768 V=30.0 PL=1
MOVL C00769 V=30.0 PL=1
MOVL C00770 V=30.0 PL=1
MOVL C00771 V=30.0 PL=1
MOVL C00772 V=30.0 PL=1
MOVL C00773 V=30.0 PL=1
MOVL C00774 V=30.0 PL=1
MOVL C00775 V=30.0 PL=1
MOVL C00776 V=30.0 PL=1
MOVL C00777 V=30.0 PL=1
MOVL C00778 V=30.0 PL=1
MOVL C00779 V=30.0 PL=1
MOVL C00780 V=30.0 PL=1
MOVL C00781 V=30.0 PL=1
MOVL C00782 V=30.0 PL=1
MOVL C00783 V=30.0 PL=1
MOVL C00784 V=30.0 PL=1
MOVL C00785 V=30.0 PL=1
MOVL C00786 V=30.0 PL=1
MOVL C00787 V=30.0 PL=1
MOVL C00788 V=30.0 PL=1
MOVL C00789 V=30.0 PL=1
MOVL C00790 V=30.0 PL=1
MOVL C00791 V=30.0 PL=1
MOVL C00792 V=30.0 PL=1
MOVL C00793 V=30.0 PL=1
MOVL C00794 V=30.0 PL=1
MOVL C00795 V=30.0 PL=1
MOVL C00796 V=30.0 PL=1
MOVL C00797 V=30.0 PL=1
MOVL C00798 V=130.0 PL=1
MOVL C00799 V=130.0 PL=1
MOVL C00800 V=30.0 PL=1
MOVL C00801 V=30.0 PL=1
MOVL C00802 V=30.0 PL=1
MOVL C00803 V=30.0 PL=1
MOVL C00804 V=30.0 PL=1
MOVL C00805 V=30.0 PL=1
MOVL C00806 V=30.0 PL=1
MOVL C00807 V=30.0 PL=1
MOVL C00808 V=30.0 PL=1
MOVL C00809 V=30.0 PL=1
MOVL C00810 V=30.0 PL=1
MOVL C00811 V=30.0 PL=1
MOVL C00812 V=30.0 PL=1
MOVL C00813 V=30.0 PL=1
MOVL C00814 V=30.0 PL=1
MOVL C00815 V=30.0 PL=1
MOVL C00816 V=30.0 PL=1
MOVL C00817 V=30.0 PL=1
MOVL C00818 V=30.0 PL=1
MOVL C00819 V=30.0 PL=1
MOVL C00820 V=30.0 PL=1
MOVL C00821 V=30.0 PL=1
MOVL C00822 V=30.0 PL=1
MOVL C00823 V=30.0 PL=1
MOVL C00824 V=30.0 PL=1
MOVL C00825 V=30.0 PL=1
MOVL C00826 V=30.0 PL=1
MOVL C00827 V=30.0 PL=1
MOVL C00828 V=30.0 PL=1
MOVL C00829 V=30.0 PL=1
MOVL C00830 V=30.0 PL=1
MOVL C00831 V=30.0 PL=1
MOVL C00832 V=30.0 PL=1
MOVL C00833 V=30.0 PL=1
MOVL C00834 V=30.0 PL=1
MOVL C00835 V=30.0 PL=1
MOVL C00836 V=30.0 PL=1
MOVL C00837 V=30.0 PL=1
MOVL C00838 V=30.0 PL=1
MOVL C00839 V=30.0 PL=1
MOVL C00840 V=30.0 PL=1
MOVL C00841 V=30.0 PL=1
MOVL C00842 V=30.0 PL=1
MOVL C00843 V=30.0 PL=1
MOVL C00844 V=30.0 PL=1
MOVL C00845 V=30.0 PL=1
MOVL C00846 V=30.0 PL=1
MOVL C00847 V=30.0 PL=1
MOVL C00848 V=30.0 PL=1
MOVL C00849 V=30.0 PL=1
MOVL C00850 V=30.0 PL=1
MOVL C00851 V=30.0 PL=1
MOVL C00852 V=30.0 PL=1
MOVL C00853 V=30.0 PL=1
MOVL C00854 V=30.0 PL=1
MOVL C00855 V=30.0 PL=1
MOVL C00856 V=30.0 PL=1
MOVL C00857 V=30.0 PL=1
MOVL C00858 V=30.0 PL=1
MOVL C00859 V=30.0 PL=1
MOVL C00860 V=30.0 PL=1
MOVL C00861 V=30.0 PL=1
MOVL C00862 V=30.0 PL=1
MOVL C00863 V=30.0 PL=1
MOVL C00864 V=30.0 PL=1
MOVL C00865 V=30.0 PL=1
MOVL C00866 V=30.0 PL=1
MOVL C00867 V=30.0 PL=1
MOVL C00868 V=30.0 PL=1
MOVL C00869 V=30.0 PL=1
MOVL C00870 V=30.0 PL=1
MOVL C00871 V=30.0 PL=1
MOVL C00872 V=30.0 PL=1
MOVL C00873 V=30.0 PL=1
MOVL C00874 V=30.0 PL=1
MOVL C00875 V=30.0 PL=1
MOVL C00876 V=30.0 PL=1
MOVL C00877 V=30.0 PL=1
MOVL C00878 V=30.0 PL=1
MOVL C00879 V=30.0 PL=1
MOVL C00880 V=30.0 PL=1
MOVL C00881 V=30.0 PL=1
MOVL C00882 V=30.0 PL=1
MOVL C00883 V=30.0 PL=1
MOVL C00884 V=130.0 PL=1
MOVL C00885 V=130.0 PL=1
MOVL C00886 V=30.0 PL=1
MOVL C00887 V=130.0 PL=1
MOVL C00888 V=130.0 PL=1
MOVL C00889 V=30.0 PL=1
MOVL C00890 V=130.0 PL=1
MOVL C00891 V=60.0 PL=1
MOVL C00892 V=60.0 PL=1
MOVL C00893 V=60.0 PL=1
MOVL C00894 V=60.0 PL=1
MOVL C00895 V=130.0 PL=1
MOVL C00896 V=30.0 PL=1
MOVL C00897 V=30.0 PL=1
MOVL C00898 V=30.0 PL=1
MOVL C00899 V=30.0 PL=1
MOVL C00900 V=30.0 PL=1
MOVL C00901 V=30.0 PL=1
MOVL C00902 V=30.0 PL=1
MOVL C00903 V=30.0 PL=1
MOVL C00904 V=130.0 PL=1
MOVL C00905 V=130.0 PL=1
MOVL C00906 V=30.0 PL=1
MOVL C00907 V=130.0 PL=1
MOVL C00908 V=30.0 PL=1
MOVL C00909 V=130.0 PL=1
MOVL C00910 V=30.0 PL=1
MOVL C00911 V=130.0 PL=1
MOVL C00912 V=20.0 PL=1
MOVL C00913 V=130.0 PL=1
MOVL C00914 V=130.0 PL=1
MOVL C00915 V=30.0 PL=1
MOVL C00916 V=130.0 PL=1
MOVL C00917 V=60.0 PL=1
MOVL C00918 V=60.0 PL=1
MOVL C00919 V=60.0 PL=1
MOVL C00920 V=60.0 PL=1
MOVL C00921 V=130.0 PL=1
MOVL C00922 V=30.0 PL=1
MOVL C00923 V=30.0 PL=1
MOVL C00924 V=30.0 PL=1
MOVL C00925 V=30.0 PL=1
MOVL C00926 V=30.0 PL=1
MOVL C00927 V=30.0 PL=1
MOVL C00928 V=30.0 PL=1
MOVL C00929 V=30.0 PL=1
MOVL C00930 V=130.0 PL=1
MOVL C00931 V=130.0 PL=1
MOVL C00932 V=30.0 PL=1
MOVL C00933 V=130.0 PL=1
MOVL C00934 V=30.0 PL=1
MOVL C00935 V=130.0 PL=1
MOVL C00936 V=30.0 PL=1
MOVL C00937 V=130.0 PL=1
MOVL C00938 V=20.0 PL=1
MOVL C00939 V=130.0 PL=1
MOVL C00940 V=130.0 PL=1
MOVL C00941 V=30.0 PL=1
MOVL C00942 V=130.0 PL=1
MOVL C00943 V=60.0 PL=1
MOVL C00944 V=60.0 PL=1
MOVL C00945 V=60.0 PL=1
MOVL C00946 V=60.0 PL=1
MOVL C00947 V=130.0 PL=1
MOVL C00948 V=30.0 PL=1
MOVL C00949 V=30.0 PL=1
MOVL C00950 V=30.0 PL=1
MOVL C00951 V=30.0 PL=1
MOVL C00952 V=30.0 PL=1
MOVL C00953 V=30.0 PL=1
MOVL C00954 V=30.0 PL=1
MOVL C00955 V=30.0 PL=1
MOVL C00956 V=130.0 PL=1
MOVL C00957 V=130.0 PL=1
MOVL C00958 V=30.0 PL=1
MOVL C00959 V=130.0 PL=1
MOVL C00960 V=30.0 PL=1
MOVL C00961 V=130.0 PL=1
MOVL C00962 V=30.0 PL=1
MOVL C00963 V=130.0 PL=1
MOVL C00964 V=20.0 PL=1
MOVL C00965 V=130.0 PL=1
MOVL C00966 V=130.0 PL=1
MOVL C00967 V=30.0 PL=1
MOVL C00968 V=130.0 PL=1
MOVL C00969 V=60.0 PL=1
MOVL C00970 V=60.0 PL=1
MOVL C00971 V=60.0 PL=1
MOVL C00972 V=60.0 PL=1
MOVL C00973 V=130.0 PL=1
MOVL C00974 V=30.0 PL=1
MOVL C00975 V=30.0 PL=1
MOVL C00976 V=30.0 PL=1
MOVL C00977 V=30.0 PL=1
MOVL C00978 V=30.0 PL=1
MOVL C00979 V=30.0 PL=1
MOVL C00980 V=30.0 PL=1
MOVL C00981 V=30.0 PL=1
MOVL C00982 V=130.0 PL=1
MOVL C00983 V=130.0 PL=1
MOVL C00984 V=30.0 PL=1
END
